	OUT_SetptQ					: REAL; 		(* (kVAr) Reactive power setpoint *)
	OUT_SetptQMax				: REAL;			(* (kVAr) Upper range of the Reactive Power setpoint*)
	OUT_SetptQMin				: REAL;			(* (kVAr) Lower range of the Reactive Power setpoint*)

	OUT_CmdReset				: BOOL ; 		(* (NA) Reset Command *) 
	
	MesHeartbeat				: BOOL ;		(*	NA) Heartbit of PCS*)
	MesCP_Read					: BOOL := TRUE;	(* (NA) CP to read values from PCS*)
	MesCP_Write					: BOOL := TRUE;	(* (NA) CP to write values from PCS*)
	
	
END_STRUCT
END_TYPE

// ---- 01_Equipement_Library/PCS/PCS_Sma.TcDUT
TYPE PCS_Sma :
STRUCT
		MesData					: PCS;		(* (NA) INV Struct*)
  	
	// System Parameter
		MesID_SystemState		:UINT; (* (-) Operating command for battery inverter, specified externally [AuxCtl.SCSOpCm d] *)
	
	// System Settings 
		MesID_CmdStopSystem		:UINT; (* (-) Disconnection of the inverter [FstStop] *)
		MesSetptQ_hldreg		:REAL; (* (%) Reactive power setpoint Q, in % of the maximum reactive power (with regard to VArRtg) of the inverter. [VArSpt] *)
		MesSetptP_hldreg		:REAL; (* (%) Active power setpoint P, in % of the maximum active power [WSpt] *)
	
	// inverter parameter
		MesID_CmdStop			:UINT; (* (-) Operating state of the inverter, setpoint [InvOpMod] *)
		MesErrClr				:UINT; (* (-) Acknowledgment of the present error [ErrClr] *)
		MesErrClrProErr			:UINT; (* (-) Acknowledging of safety-relevant errors [ErrClr.ProErr] *)
								
	// INV Measures 
		MesIdcStk1				:REAL; (* (A) DC current inverter bridge 1 [DcMs.Amp.Stk1] *)
		MesIdcStk2				:REAL; (* (A) DC current inverter bridge 2 [DcMs.Amp.Stk2] *)
		MesIdcStk3				:REAL; (* (A) DC current inverter bridge 3 [DcMs.Amp.Stk3] *)
		MesUdcStk1				:REAL; (* (V) DC voltage of the inverter bridge 1 [InvMs.DclVol.Stk1] *)
		MesUdcStk2				:REAL; (* (V) DC voltage of the inverter bridge 2 [InvMs.DclVol.Stk2] *)
		MesUdcStk3				:REAL; (* (V) DC voltage of the inverter bridge 3 [InvMs.DclVol.Stk3] *)
		MesIacL1				:REAL; (* (A) AC current L1, total [InvMs.TotA.PhsA] *)
		MesIacL2				:REAL; (* (A) AC current L2, total [InvMs.TotA.PhsB] *)
		MesIacL3				:REAL; (* (A) AC current L3, total [InvMs.TotA.PhsC] *)
		MesU12					:REAL; (* (V) Line-to-line voltage L1-L2, utility grid [GriMs.V.PhsAB] *)
		MesU23					:REAL; (* (V) Line-to-line voltage L2-L3, utility grid [GriMs.V.PhsBC] *)
		MesU31					:REAL; (* (V) Line-to-line voltage L3-L1, utility grid [GriMs.V.PhsCA] *)
		MesTmpAcCab				:REAL; (* (°C) Temperature in the AC range [TmpCab.Acc] *)
		MesTmpDcCab				:REAL; (* (°C) Temperature in the DC range [TmpCab.Dcc] *)
		MesTmpRioCab			:REAL; (* (°C) Temperature in the electronics area [TmpCab.Rio] *)
		MesTmpMax				:REAL; (* (°C) Temperature in interior, maximum value [TmpCab.Max] *)
		MesTmpIgbtMax			:REAL; (* (°C) Temperature of the inverter bridge (switch), maximum value [TmpStk.IgbtMax] *)
		MesTmpPcbMax			:REAL; (* (°C) Temperature of the inverter bridge (assembly), maximum value [TmpStk.PcbMax] *)
		MesTmpExt				:REAL; (* (°C) External temperature [TmpExl] *)
		MesTmpTransfo			:REAL; (* (°C) Temperature of the MV transformer [TmpTrf] *)
		MesID_SttDcSw1			:UINT; (* (-) Switching status of the DC load-break switch 1 [DcSw1Stt] *)
		MesID_SttDcSw2			:UINT; (* (-) Switching status of the DC load-break switch 2 [DcSw2Stt] *)
		MesID_SttDcSw3			:UINT; (* (-) Switching status of the DC load-break switch 3 [DcSw3Stt] *)
		MesID_SttAcSw			:UINT; (* (-) Switching status of the AC circuit breaker [AcSwStt] *)
		MesID_SttCapac			:UINT; (* (-) Switching state of the capacitor contactor [CapacSwStt] *)
		MesID_SttPrchrg			:UINT; (* (-) Switching status of the pre- charging contactor [PrchrgSwStt] *)
		MesEdcTot				:REAL; (* (MWh) DC energy drawn, total [Cnt.TotDcWhIn] *)
		MesEacTot				:REAL; (* (MWh) AC energy fed in, total [Cnt.TotAcWhOut] *)
		MesEdcDay				:REAL; (* (MWh) DC energy drawn that day [Cnt.DcWhIn] *)
		MesEacDay				:REAL; (* (MWh) AC energy fed in that day [Cnt.AcWhOut] *)
		MesID_ErrLcn			:UINT; (* (-) Error location of the present error [ErrLcn] *)
		MesID_ErrStt			:UINT; (* (-) Error status of the inverter [ErrStt] *)
		MesNum_Err				:UINT; (* (-) Error number of the present error [ErrNo] *)
		MesID_SttKey			:UINT; (* (-) Switch status of the start-stop key switch [Rio.KeySw] *) 
		MesTime_Feed			:UINT; (* (s) Feed-in time [Cnt.TotFeedTm] *)
		MesTime_Run				:UINT; (* (s) Operating time [Cnt.TotOpTm] *)
		MesTime_Fan1			:UINT; (* (s) Operating time of the interior fan 1 [Cnt.FanCab1Tm] *)
		MesTime_Fan2			:UINT; (* (s) Operating time of the interior fan 2 [Cnt.FanCab2Tm] *)
		MesTime_StkFan			:UINT; (* (s) Operating time of the inverter bridge fan [Cnt.FanStkTm] *)
		MesTime_Heater			:UINT; (* (s) Operating time of the interior heater [Cnt.HtCabTm] *)
		MesTime_Heater40C		:UINT; (* (s) Operating time of the -40°C interior heater [Cnt.HtLoExlTmpTm] *)
		MesTimeWait_Grid		:UINT; (* (s) Waiting time for grid connection [WaitGriTm] *)
		MesSerial				:UINT; (* (-) Inverter serial number [DevInf.SerNo] *)
		MesID_SttGfdi			:UINT; (* (-) Switching status of the GFDI [GfdiSwStt] *)
		MesSetptP				:REAL; (* (kW) Active power, setpoint [WSpt] *)
		MesSetptSmax			:REAL; (* (kVA) Maximum apparent power, setpoint [VAMaxSpt] *)
		MesSetptQ				:REAL; (* (kVAr) Reactive power, setpoint [VArSpt] *)
		MesCosPhisetpt			:REAL; (* (-) Power factor cos (phi), setpoint [PFSpt] *)
		MesID_SttPresTransfo	:UINT; (* (-) Fast stop hermetic protection, pressure [TrfPro.Pres] *)
		MesID_SttTempAlarmTransfo:UINT; (* (-) Fast stop hermetic protection, temperature [TrfPro.TmpTrp] *)
		MesID_SttOilAlarmTransfo:UINT; (* (-) Hermetic protection, gas fill level [TrfPro.GasOilLev] *)
		MesID_SttTempWarnTransfo:UINT; (* (-) Hermetic pressure, temperature warning [TrfPro.TmpWrn] *)
		MesTmpStk1				:REAL; (* (°C) Temperature of inverter bridge 1 (switch) [TmpStk1.lgbt] *)
		MesTmpStk2				:REAL; (* (°C) Temperature of inverter bridge 2 (switch) [TmpStk2.lgbt] *)
		MesTmpStk3				:REAL; (* (°C) Temperature of inverter bridge 3 (switch) [TmpStk3.lgbt] *)
		MesTmpStk1Max			:REAL; (* (°C) Maximum temperature of inverter bridge 1 (assembly) [TmpStk1.Pcb] *)
		MesTmpStk2Max			:REAL; (* (°C) Maximum temperature of inverter bridge 2 (assembly) [TmpStk2.Pcb] *)
		MesTmpStk3Max			:REAL; (* (°C) Maximum temperature of inverter bridge 3 (assembly) [TmpStk3.Pcb] *)
		MesEacPrevDay			:REAL; (* (MWh) AC energy fed in the previous day [Cnt.YstdWhOut] *)
		MesTime_CPU				:REAL; (* (s) CPU running time since system start [Cpu1UpTime] *)
		MesRiso					:REAL; (* (kOhm) Insulation resistance [PvGnd.RisIso] *)
		MesPressureTransfo		:REAL; (* (-) MV transformer pressure [PresTrf] *)
		MesID_SttPressureSensor	:UINT; (* (-) Error status of MV transformer pressure monitoring [PresTrf.ErrStt] *)
		MesSetptPmax			:REAL; (* (pu) Available Active Power [WAval] *)
		MesSetptQmax			:REAL; (* (pu) Available reactive power [VArAval] *)
		MesID_SttDrt			:UINT; (* (-) Current derating status [DrtStt] *)
		MesID_PwrOffReas		:UINT; (* (-) Current cause of inverter disconnection [PwrOffReas] *)
		MesPnom_stpt			:REAL; (* (kW) Nominal value of active power [WRtg] *)
		MesActErrNo1			:UINT; (* (-) Error number of the current error [ActErrNo1] *)
		MesActErrLcn1			:UINT; (* (-) Location where the current error was detected [ActErrLcn1] *)
		MesActErrNo2			:UINT; (* (-) Error number of the current error [ActErrNo2] *)
		MesActErrLcn2			:UINT; (* (-) Location where the current error was detected [ActErrLcn2] *)
		MesActErrNo3			:UINT; (* (-) Error number of the current error [ActErrNo3] *)
		MesActErrLcn3			:UINT; (* (-) Location where the current error was detected [ActErrLcn3] *)
		MesActErrNo4			:UINT; (* (-) Error number of the current error [ActErrNo4] *)
		MesActErrLcn4			:UINT; (* (-) Location where the current error was detected [ActErrLcn4] *)
		MesActErrNo5			:UINT; (* (-) Error number of the current error [ActErrNo5] *)
		MesActErrLcn5			:UINT; (* (-) Location where the current error was detected [ActErrLcn5] *)
		MesActErrNo6			:UINT; (* (-) Error number of the current error [ActErrNo6] *)
		MesActErrLcn6			:UINT; (* (-) Location where the current error was detected [ActErrLcn6] *)
		MesActErrNo7			:UINT; (* (-) Error number of the current error [ActErrNo7] *)
		MesActErrLcn7			:UINT; (* (-) Location where the current error was detected [ActErrLcn7] *)
		MesActErrNo8			:UINT; (* (-) Error number of the current error [ActErrNo8] *)
		MesActErrLcn8			:UINT; (* (-) Location where the current error was detected [ActErrLcn8] *)
		MesActErrNo9			:UINT; (* (-) Error number of the current error [ActErrNo9] *)
		MesActErrLcn9			:UINT; (* (-) Location where the current error was detected [ActErrLcn9] *)
		MesActErrNo10			:UINT; (* (-) Error number of the current error [ActErrNo10] *)
		MesActErrLcn10			:UINT; (* (-) Location where the current error was detected [ActErrLcn10] *)
		MesQref_stptExt			:REAL; (* (kVAr) Reference value for the external reactive power setpoint [VArExlSpt.RefVal] *)
		MesPref_stptExt			:REAL; (* (kW) Reference value for the external active power setpoint [WExlSpt.RefVal] *)
		ModbusValue 			:WORD;
		MesQref_stpt			:REAL; (* (kvar) Nominal value of reactive power [VArRtg] *)
		MesUdc_plusGnd			:REAL; (* (V) DC voltage of DC+ to ground [DcMs.VolPosGnd] *)
		MesUdc_minusGnd			:REAL; (* (V) DC voltage of DC- to ground [DcMs.VolNegGnd] *)
		MesID_State_Imax		:UINT; (* (-) Overload capability: Overcurrent status [GriForm.OvAmpStt] *)
		MesTimeWait_Error		:REAL; (* (s) Remaining error waiting period [ErrRmgTm] *)
		
	// State ID 
		MesID_OpeMode			: WORD ; (* SMA Operating Mode  ENUM *)
		MesID_OpStt				: WORD ; (* SMA Operation State ENUM *)
		MesID_OpeProErr			: WORD ; (* SMA Saftey Error  ENUM *)
		MesID_ErrClr			: WORD ; (* SMA Error ENUM *)

	// Output 
		OUT_CmdReset_Safety		: BOOL ;(* Safety reset ordered *) 
		OUT_CmdOpenAC			: BOOL ; (* Open AC Command*)
END_STRUCT
END_TYPE

// ---- 01_Equipement_Library/PCS/PCS_Jema_IBX3.TcDUT
///////////
// Structure for CtrlPcs Jema .  
//////////
TYPE PCS_Jema_IBX3 :
STRUCT
// PCS Controller  Measures
	AX_PowerCol					: ARRAY[1..3] OF PowerCol_Jema;

	MesData						: PCS ; 
	
	
	MesNbPowerCol_FreqReg			: UINT  ; (*(NA) Number of Power Column doing frequency regulation *)
	MesState_SoCLimitReached		: BOOL ; (*(NA) PCS SoC Limits has been reached *)
	MesHumidity						: REAL ; (*(%) Humidity*)
	
	MesReadCompleted				: BOOL ; 
	
	OUT_CmdBlackStart			: BOOL ; (* (NA) Blackstart Command *) 
	OUT_CmdGridMode				: BOOL ; (* (NA) Grid Mode Command *) 
	OUT_CmdP					: BOOL ; (* (NA) P setpoint regulation Mode Command *) 
	
	OUT_CmdQ				: BOOL ; (* (NA) Q setpoint regulation Mode Command *) 
	OUT_SetptV				: REAL ; (* (V) Voltage Reference for offgrid Mode *) 
	OUT_SetptCosPhi			: REAL ; (* (p.u) Cosphi Reference for Cosphi reg Mode *) 
	
	OUT_SetptF				: REAL ; 	(* (Hz) Frequency Reference for offgrid Mode *) 
	OUT_CmdCosPhi			: BOOL ; (* (NA) Cosphi regulation Mode Command *) 
	OUT_CmdUregMode			: BOOL ; (* (NA) Voltage Regulation Mode Command *) 
	OUT_CmdFreqregMode	: BOOL ; (* (NA) Frequency Regulation Mode Command *) 
END_STRUCT
END_TYPE

// ---- 01_Equipement_Library/PCS/PCS_PE.TcDUT
{attribute 'pack_mode' := '1'}
TYPE PCS_PE :
STRUCT
// PCS Controller  Measures
	AX_PowerCol					: ARRAY[1..6] OF PowerCol_PE;		(* PE Module*)
	
	MesData						: PCS ; (* MesData*)
	
	MesP_ChargeMax				: REAL ;		(* (%)	Max active power setpoint. SV4.2.1a	*)
	MesP_DischargeMax			: REAL ;		(* (%)	Max active power setpoint. SV4.2.1b	*)
	MesP_ChargeMax1				: REAL ;		(* (%)	Max active power setpoint1. SV4.2.1a	*)
	MesP_DischargeMax1			: REAL ;		(* (%)	Max active power setpoint1. SV4.2.1b	*)
	MesP_ChargeMax2				: REAL ;		(* (%)	Max active power setpoint2. SV4.2.1a	*)
	MesP_DischargeMax2			: REAL ;		(* (%)	Max active power setpoint2. SV4.2.1b	*)
	
	//Electrical Measurements	
	MesI1						: REAL; (* (A) Current phase 1 (R). INV: SV1.4 Grid current I1 (HEMK)															*)
	MesI2						: REAL; (* (A) Current phase 2 (S). INV: SV1.5 Grid current I2 (HEMK)															*)
	MesI3						: REAL; (* (A) Current phase 3 (T). INV: SV1.6 Grid current I3  (HEMK)															*)
	MesU12						: REAL; (* (V) Phase AB RMS voltage (line to line)at grid side of AC circuit breaker CB501. INV: SV1.1 Grid voltage RS (HEMK)	*)
	MesU23						: REAL; (* (V) Phase BC RMS voltage (line to line)at grid side of AC circuit breaker CB501. INV: SV1.2 Grid voltage ST(HEMK)	*)
	MesU31						: REAL; (* (V) Phase CA RMS voltage (line to line)at grid side of AC circuit breaker CB501. INV: SV1.3 Grid voltage TR (HEMK)	*)

	MesHumidity					: REAL;			(* (%) Humidity sensor	*)
	MesPconnected				: REAL; (* (%) Current available active power. INV: SV4.1.2 P limit inst 														*)  
	MesQconnected				: REAL; (* (%) Current available reactive power. INV: SV4.2.2 Q limit inst 														*)                                                      									

	MesIDState_InsuResistor_DC	: WORD ; (* (NA) Status of insulation protection. 0 = Idle, 1= Inter measurement quard, 2=measurement in progress, 3=self-test in progress, 4=risk addressed state SV3.1.1 *)
	MesInsuResistor_AC			: REAL;	(* (Ohms) AC Insulation Resistance. INV: SV3.1.2  Resistor 																*)
	MesIDState_InsuResistor_AC	: WORD ; (* (NA) Status of insulation protection. 0 = Idle, 1= Inter measurement quard, 2=measurement in progress, 3=self-test in progress, 4=risk addressed state SV3.1.1 *)
	MesInsuResistor_DC			: REAL;	(* (Ohms) DC Insulation Resistance. INV: SV3.2.2  Resistor 		*)
	MesInsuResistor_DC2			: REAL; (* (Ohms) DC Insulation Resistance. INV: SV3.3.2  Resistor 		*)

	MesUdc_Input1		 		: REAL ; (* (V) DC Voltage Bus 1 . INV : SV2.1.1 *)
	MesUdc_Input2		 		: REAL ; (* (V) DC Voltage Bus 2 . INV : SV2.1.2*)
	MesUdc_Input3		 		: REAL ; (* (V) DC Voltage Bus 3 . INV : SV2.1.3*)
	MesUdc_Bat1		 			: REAL ; 	(* (V) DC Voltage BESS 1 . INV : SV2.4.1*)
	MesUdc_Bat2		 			: REAL ; 	(* (V) DC Voltage BESS 2 . INV : SV2.4.2*)
	MesUdc_Bat3		 			: REAL ; 	(* (V) DC Voltage BESS 3 . INV : SV2.4.3*)
	MesPdc_Input1		 		: REAL ; (* (V) DC Power Bus 1 . INV : SV2.5a*)
	MesPdc_Input2		 		: REAL ; (* (V) DC Power Bus 2 . INV : SV2.5b*)
	MesPdc_Input3		 		: REAL ; (* (V) DC Power Bus 3 . INV : SV2.5c*)
	MesIdc_RFI_Input1    		: REAL ; (* (V) RFI Current  Bus 1 . INV : SV2.11a*)
	MesIdc_RFI_Input2    		: REAL ; (* (V) RFI Current  Bus 2 . INV : SV2.11b*)
	MesIdc_RFI_Input3	 		: REAL ; (* (V) RFI Current  Bus 3 . INV : SV2.11c*)
	MesIdc_Input1				: REAL; (*(A) SV2.6a DC input current*)
	MesIdc_Input2				: REAL; (*(A) SV2.6b DC input current*)
	MesIdc_Input3				: REAL; (*(A) SV2.6c DC input current*)

	//Status Summary
	MesIDState					: UINT; (* (NA) Current inverter status . INV : SV4.1.3                                                    *)                 	
	MesAlarmID					: WORD;	(* (NA) Alarm ID of the currently active event.  INV : SV4.1.1    *)
	MesWarningID				: WORD;	(* (NA) Warning ID of the currently active event.  INV : SV4.1.2    *)
	MesEventID					: WORD;	(* (NA) Event ID of the currently active event.  INV : SV9.1.1 :Last Event    *)
                    	
	// Inverter's Control Cabinet  Status                                                                       											
	MesTemp_IGBTmax				: REAL; 		 (* (C) Maximum IGBT temperature. INV: SV4.1.5 Max IGBTs temperature											*)
	MesTemp_PowerColmax			: REAL; 		 (* (C) Maximum power column temperature. INV: SV4.1.6 Max modules temperature									*)
 
	MesReadModule				: UINT;		(* (NA) module read *)
	MesIDState_PowerCol			: WORD ; 	(* (NA) Running modules (0 = stopped, 1 =running). Module 1 is the first from the right. SV9.1.1															*)
               	                                                   	                                						
	// Reset command        	                                                                     	                                						
	OUT_CmdReset 				: BOOL; 		 (* (NA) OUT reset command. INV: Reset command 43012															*)
	MesCalibrationState		 	: WORD;			(*(NA) it's a state to know if the calibration is ongoing or not, (0=running, 1=Discharging the batteries started, 2=20min hold finished, starting to send setpt of 0 for 20min, 3=Charging started*)
	MesBMSSelected				: WORD;
	OUT_SetptPMax_IMDicharge1	: REAL;
	OUT_SetptPMax_IMDicharge2	: REAL;
	OUT_SetptPMax_IMCharge1		: REAL;
	OUT_SetptPMax_IMCharge2		: REAL;
	MesSelector 				: BOOL;
	
	
END_STRUCT
END_TYPE

// ---- 01_Equipement_Library/PCS/PowerCol_JemaAlarms.TcDUT
TYPE PowerCol_JemaAlarms :
STRUCT

// ALARM0 bAlarm1
		MesI1_Alm			: BOOL; 	//RegAlarms0: I1_Alm
		MesI2_Alm			: BOOL; 	//RegAlarms0: I2_Alm
		MesI3_Alm			: BOOL; 	//RegAlarms0: I3_Alm
		MesVdc_High_Alm		: BOOL; 	//RegAlarms0: Vdc_High_Alm
		MesVdc_Low_Alm		: BOOL; 	//RegAlarms0: Vdc_Low_Alm
		                            	// 
		MesU12_High_Alm		: BOOL; 	//RegAlarms0: U12_High_Alm
		MesU12_Low_Alm		: BOOL; 	//RegAlarms0: U12_Low_Alm
		MesU23_High_Alm		: BOOL; 	//RegAlarms0: U23_High_Alm
		MesU23_Low_Alm		: BOOL; 	//RegAlarms0: U23_Low_Alm
		MesU31_High_Alm		: BOOL; 	//RegAlarms0: U31_High_Alm
		MesU31_Low_Alm		: BOOL; 	//RegAlarms0: U31_Low_Alm
		MesVd_High_Alm		: BOOL; 	//RegAlarms0: Vd_High_Alm
		MesVd_Low_Alm		: BOOL; 	//RegAlarms0: Vd_Low_Alm
		MesVdc_Neg			: BOOL; 	//RegAlarms0: Vdc_Neg
		                            	//   :blabla
										//wAlarmCode
		
// ALARM1 bAlarm1
		MesU1223_Unbalance	: BOOL;		//RegAlarms1: U1223_Unbalance
		MesU2331_Unbalance	: BOOL;		//RegAlarms1: U2331_Unbalance
		MesU3112_Unbalance	: BOOL;		//RegAlarms1: U3112_Unbalance
		MesInvertedPhase	: BOOL;		//RegAlarms1: InvertedPhase
		MesI12_Unbalance	: BOOL;		//RegAlarms1: I12_Unbalance
		MesI23_Unbalance	: BOOL;		//RegAlarms1: I23_Unbalance
		MesI31_Unbalance	: BOOL;		//RegAlarms1: I31_Unbalance
		MesCouplingTimeout	: BOOL;		//RegAlarms1: CouplingTimeout
		MesF_High			: BOOL;		//RegAlarms1: F_High
		MesF_Low			: BOOL;		//RegAlarms1: F_Low
		MesGrndFault		: BOOL;		//RegAlarms1: GrndFault
		MesVaristor			: BOOL;		//RegAlarms1: Varistor
		MesPcbOverTemp		: BOOL;		//RegAlarms1: PcbOverTemp
		MesHeatsinkOverTemp	: BOOL;		//RegAlarms1: HeatsinkOverTemp
		                           		// 
		MesOvertempHyst		: BOOL;		//RegAlarms1: OvertempHyst
		//wAlarmCode
// ALARM2 bAlarm1
										// 
                                    	// 
                                    	// 
                                    	// 
		MesGridCbOpened		: BOOL;		//RegAlarms2: GridCbOpened
		MesGridCbTrip		: BOOL;		//RegAlarms2: GridCbTrip
										//
		                           		// 
		MesGridContactFail	: BOOL;		//RegAlarms2: GridContactFail 
		MesDoorOpened		: BOOL;		//RegAlarms2: DoorOpened 
		                           		// 
		                           		// 
		MesVdcPrechargewrong: BOOL;		//RegAlarms2: VdcPrechargewrong 
		                           		// 
		MesOverVoltHyst		: BOOL;		//RegAlarms2: OverVoltHyst 
		MesIdcMax			: BOOL;		//RegAlarms2: IdcMax 
		//wAlarmCode
		
//ALARM3   bAlarm1                         
		MesSKIIP1			: BOOL; 	//RegAlarms3: SKIIP1
		MesSKIIP2			: BOOL; 	//RegAlarms3: SKIIP2
		MesSKIIP3			: BOOL; 	//RegAlarms3: SKIIP3
		MesSKIIP_OT			: BOOL; 	//RegAlarms3: SIIP_OT
		MesFPGA_WdogTrip	: BOOL; 	//RegAlarms3: FPGA_WdogTrip
		MesStopEverything	: BOOL; 	//RegAlarms3: StopEverything
		MesIMax				: BOOL; 	//RegAlarms3: IMax
		MesEmergencyStop	: BOOL; 	//RegAlarms3: EmergencyStop
		MesImdWarning		: BOOL; 	//RegAlarms3: ImdWarning
		MesImdFault			: BOOL; 	//RegAlarms3: ImdFault
		                            	//RegAlarms3:  
		MesCoilOverTemp		: BOOL; 	//RegAlarms3: CoilOverTemp
		                            	//RegAlarms3:  
		MesAlrmGrp1_Curr	: BOOL; 	//RegAlarms3: AlrmGrp1_Curr
		MesAlrmGrp2_Curr	: BOOL; 	//RegAlarms3: AlrmGrp2_Curr
		MesShortCircuit_DC	: BOOL; 	//RegAlarms3: ShortCircuit_DC
		//wAlarmCode
// ALARM4 bAlarm1
		MesBatError			: BOOL;		//RegAlarms4: BatError
		MesBatCtlStop		: BOOL;		//RegAlarms4: BatCtlStop
		MesBatComErrors		: BOOL;		//RegAlarms4: BatComErrors
		MesPowerUnbalance	: BOOL;		//RegAlarms4: PowerUnbalance
		MesOverpower		: BOOL;		//RegAlarms4: Overpower
		//wAlarmCode
		
END_STRUCT
END_TYPE

// ---- 01_Equipement_Library/PCS/PowerCol_Jema.TcDUT
///////////
// Structure For Jema Module 
//////////
TYPE PowerCol_Jema :
STRUCT
	
		MesData					: PowerCol ; (* MesData *) 

		MesTempControl      		: REAL ; 		// {0}(°C) Temperature of control card
		MesTempPowerUnit    		: REAL ;		// {0}(°C) Temperature of Power Unit
		MesTempCabinet      		: REAL ; 		// {0}(°C) Cabinet temperature
		MesTempCoil1        		: REAL ; 		// {0}(°C) Coil temperature
		MesRegAlarm0        		: WORD ; 		// {0}Alarm Word of PCS
		MesRegAlarm1        		: WORD ; 		// {0}Alarm Word of PCS 
		MesRegAlarm2        		: WORD ; 		// {0}Alarm Word of PCS 
		MesRegAlarm3        		: WORD ;  		// {0}Alarm Word of PCS
		MesRegAlarm4        		: WORD ;  		// {0}Alarm Word of PCS
		MesDeratingWord				: WORD ;		// {0}Derating word of PCS
		MesHeartbit					: REAL ;		// {0}Heartbit
		MesDoorOpened				: BOOL ;		// {1}Door of the Power module is opened	
		
		MesJemaAlarms				: PowerCol_JemaAlarms;

			

END_STRUCT
END_TYPE

// ---- 01_Equipement_Library/PCS/PowerCol.TcDUT
///////////
// Structure For Jema Module 
//////////
TYPE PowerCol :
STRUCT
		MesP 						: REAL; 		// {1}(kW) Active Power output (AC) of PCS
		MesQ 						: REAL; 		// {1}(kVAr) Reactive AC Power Produced by PCS 
		MesPdc						: REAL ; 		// {1}(kW) DC Power . 
		MesCosPhi 					: REAL;  		// {0}(p.u) Power factor
		MesFreq						: REAL ; 		// {0}(Hz) Frequency
		MesTemp						: REAL ; 		// {0}(°C) PCS Internal Temperature
		MesU 						: REAL;  		// {0}(V) AC Voltage measure
		MesUdc 						: REAL;  		// {0}(V) DC Voltage measure
		MesI 						: REAL; 		// {0}(A) Total AC current 
		MesI1						: REAL ; 		// {0}(A) Phase 1 AC Current
		MesI2						: REAL ;        // {0}(A) Phase 2 AC Current
		MesI3						: REAL ;        // {0}(A) Phase 3 AC Current
		MesIdc 						: REAL; 		// {0}(A) Total DC current from batteries (+ = discharge)
		MesPavailable 				: REAL;  		// {1}(kW) Available PCS Power 
		MesPconnected				: REAL ; 		// {0}(kW) Connected PCS Power 
		MesDcSwitchClosed			: BOOL ; 		// {0}(NA) Position of the DC Switch : True = Switch closed
		MesAcSwitchClosed			: BOOL ; 		// {0}(NA) Position of the AC Switch : True = Switch closed
	

			

END_STRUCT
END_TYPE

// ---- 01_Equipement_Library/PCS/PowerCol_PE.TcDUT
///////////
// Structure For Jema Module 
//////////
TYPE PowerCol_PE :
STRUCT
		
		MesData					: PowerCol ; (* MesData *) 

		AX_DCInputs			: ARRAY[1..10] OF  DCInputs_PE ;(* Object *) 
		
		MesIDState			: DWORD ;		(* (NA) 	Module status (SV9.3 PE documentation p.97)																*)
		MesTempmax			: REAL ;		(* (C) 		Maximum IGBT temperature of the selected module															*)
		MesStateIO			: WORD ;		(* (NA) 	0: Open, 1: Closed. Bit 1 =  fan contactor, Bit 2 = main AC contactor, Bit 3 = AC soft charge contactor, Bit 4 = LCL filter contactor, Bit 5 = DC contactor , Bit 6 = reserved, Bit 7 = if open : overheating in the coil, Bit 8 = fan contactor feedback, Bit 9 = AC main contactor feedback, Bit 10 = AC soft charge contactor feedback, Bit 11 = LCL filter contactor feedback , Bit 12 = DC contactor feedback *) 		
		MesHygro			: REAL ; 		(* (%) 		Percentage of humidity																					*)
		MesAlarmID			: BYTE ; 		(* (NA)  PowerColumn Alarm ID  . W65 to W116  *)
			

END_STRUCT
END_TYPE

// ---- 01_Equipement_Library/PPC/PPC.TcDUT
///////////
// Structure For Inverter. Main Operating Data to be saved ( ex: OPC ) .  
//////////
TYPE PPC :
STRUCT
	
		// INV Measures
		
		MesAlarmCom					: BOOL; 		(* (NA) PPC  Communication fault*)
		

		
		MesSetptP			: REAL;
		MesSetptQ			: REAL;		
		MesP				: REAL;
		MesQ				: REAL;

		MesNbInvAvail		: REAL;


		
		MesWatchdog			: REAl;
		CalState			: BYTE;
		
		MesCP_Read			: BOOL := TRUE;	(* (NA) Cal : Permanent Condition for Read			  *)
		MesCP_Write			: BOOL := FALSE;(* (NA) Cal : Permanenent Condition for Write	  	  *)
		   
		MesAlarmCode		: WORD ;    (* (NA) Internal Akuo AlarmCode*)
		MesWarningCode		: WORD ;    (* (NA) Internal Akuo WarningCode*)
		MesEventCode		: WORD ;    (* (NA) Internal Akuo EventCode*)
		
END_STRUCT
END_TYPE

// ---- 01_Equipement_Library/PPC/PPC_Sma.TcDUT
///////////
// Structure For Inverter. Main Operating Data to be saved ( ex: OPC ) .  
//////////
TYPE PPC_Sma :
STRUCT
	
		// INV Measures
		MesData		: PPC ; 
		
		
		MesPState			: REAL;
		MesQState			: REAL;
		MesGeneState		: REAL;

		MesPNomControlled	: REAL;
		MesPControlled		: REAL;
		MesQnomControlled	: REAL;
		MesQControlled		: REAL;
		
		
END_STRUCT
END_TYPE

// ---- 01_Equipement_Library/PPC/PPC_PE.TcDUT
TYPE PPC_PE :
STRUCT
		MesData 								: PPC;   			    (* (NA) MesData				 *)
		                                                                
		PM										: PM_PM5XXX;	    (* (NA) PM13EH PLUS			 *)
		EL3453									: PM_Standard;		    (* (NA) Beckhoff card EL3453 *)
		MesState								: UINT;				    (* (NA) PPC status. 0: PPC off and not sending commands to inverters, 1: PPC on and sending commands to inverters, 2: PPC on frequency event. 3: PPC in LVRT event. 4: PPC in HVRT event. 5, 6: Reserved *)
                                                                        	                                                            
		// Q Regulation                                                                                                                                            		    		
		ParamQfUQmin							: REAL := -5000;	    (* (kVAr) Voltage Regulation Minimal Reactive Power @ maximal voltage*) 		
		ParamQfUQmax							: REAL := 5000;  	    (* (kVAr) Voltage Regulation Maximal Reactive Power @ minimal voltage*)    		
		ParamQfUUHigh							: REAL := 25000; 	    (* (V)    Voltage Regulation Maximal voltage*)    		
		ParamQfUDdBandHigh						: REAL := 22000; 	    (* (V)    Voltage Regulation Deadband High voltage*)     		
		ParamQfUDdBandLow						: REAL := 18000; 	    (* (V)    Voltage Regulation Deadband Low voltage*)      	
		ParamQfUULow							: REAL := 15000; 	    (* (V)    Voltage Regulation Minimal Voltage*)
		MesAlarmPower							: BOOL; 				(* (NA)   Power alarm due to circuit breaker open										 						*)			
                                                                                                                                                			 							
	// PI active power                                                                                                                          			 							
		//IN_CmdPIDP_LocalMode 					: BOOL;                                                                                         			 							
		IN_SetptP_PR_Cent						: REAL;					(* (%)  Active power reference  														 						*)
		IN_SetptP_PR_MW							: REAL;					(* (MW) Active power reference 														 							*)	
		IN_Feedback_PR_Cent						: REAL;					(* (%)	Active power PI feedback 													 							*)
		IN_Feedback_PR_MW						: REAL;					(* (MW)	Active power PI feedback 													 							*)
		MesStateOL_PR							: BOOL;					(* (NA) Open loop activation of P control. 1= Open loop activated					 							*)
		IN_PIDP_SetptPOpenloop					: REAL;		            (* *)                            	                                    			 							                                                              			 
		ParamKp_PR								: REAL;					(* (NA) Kp for P regulation 														 							*)
		ParamKi_PR								: REAL;					(* (NA) Ki for P regulation 	 													 							*)
	   	ParamPIDP_Inversion						: BOOL;					(* (NA) PI inversion of active power control 										 							*)    
		ParamPID_PR_Min							: REAL; 				(* (kW) Low limit for PI for active power regulation	   							 							*)     		
		ParamPID_PR_Max							: REAL;  				(* (kW) High limit for PI for active power regulation 								 							*)          		
	    OUT_SetpointP_PR						: REAL;					(* (p.u) Active Power PI output per unit 											 							*)                                                                                                                                       			 
	
// PI frequency control                                                                                                                     			 							
		IN_SetptFreq_FR_Unit					: REAL;					(* (p.u) Frequency regulation (FR) reference  										 							*)
		IN_SetptFreq_FR_MW						: REAL;					(* (MW) Frequency regulation (FR) reference 										 							*) 
		IN_Feedback_FR_Unit						: REAL;					(* (p.u) Frequency regulation (FR) PI feedback 										 							*)
		IN_Feedback_FR_MW						: REAL;					(* (MW)	Frequency regulation (FR) PI feedback 										 							*)	
        ParamKp_FR								: REAL;					(* (NA) Kp for frequency regulation													 							*)
		ParamKi_FR								: REAL;					(* (NA) Ki for frequency regulation 		 										 							*)
	    ParamFreqnom							: REAL;					(* (NA) Nominal frequency for frequency response									 							*) 
		ParamStatism_OverFreq_Primary			: REAL; 				(* (NA) Slope for the Primary point Over Frequency in Frequency Response			 							*) 
		ParamStatism_OverFreq_Secundary			: REAL;					(* (NA) Slope for the Secundary point Over Frequency in Frequency Response 			 							*)
        ParamStatism_UnderFreq_Primary			: REAL; 				(* (NA) Slope for the Primary point under Frequency in Frequency Response			 							*) 
		ParamStatism_UnderFreq_Secundary		: REAL;					(* (NA) Slope for the Secundary point under Frequency in Frequency Response 		 							*)
		ParamDeltaPmax_OverFR					: REAL; 				(* (kW) Maximum power to be injected during under frequency regulation 		 		 							*)
        ParamDeltaPmax_UnderFR					: REAL; 				(* (kW) Maximum power to be reduced during over frequency regulation 		 		 							*)
		ParamDeadBand_FR						: REAL;					(* (mHz) Frequency regulation dead band axis Y										 							*) 
		MesEventID_FR							: UINT;					(* (NA) Frequency Response Event State. 0: No Event, 1: Over Frequency Primary Band, 2: Over Frequency Secondary Band, 3: Over Frequency Terciary Band, 4: Under Frequency Primary Band, 5: Under Frequency Secondary Band, 6: Under Frequency Terciary Band *)
 		MesStateID_FR							: BOOL;					(* (NA) Frequency Mode Selector. Calculation basis: 0: unitary base, 1: Power freeze 							*)		
		MesState_FR								: BOOL;					(* (NA) Activation/deactivation of frequency regulation. 1= activated				 							*)
		                               
	// PID Q direct                               	
		IN_SetptQ_QR_Cent					    : REAL;					(* (%) Reactive power reference  													 							*)
		IN_SetptQ_QR_MW							: REAL;					(* (MVAr) Reactive power reference 													 							*)	
		IN_Feedback_QR_Cent						: REAL;					(* (%) Reactive power PI feedback 													 							*)
		IN_Feedback_QR_MW						: REAL;					(* (MVAr) Reactive power PI feedback 												 							*)
		MesStateOL_QR							: BOOL;					(* (NA) Open loop activation of Q control. 1= Open loop activated					 							*)
		ParamKp_QR								: REAL;					(* (NA) Kp pour régulation Q 										 				 							*)
		ParamKi_QR								: REAL; 				(* (NA) Ki pour régulation Q 														 							*)
 		ParamPID_QR_Min							: REAL; 				(* (kVAr) Low limit for PID of reactive Power  										 							*)     		
		ParamPID_QR_Max							: REAL;  				(* (kVAr) High limit for PID of active Power										 							*)
		ParamPIDQ_Inversion						: BOOL;					(* (NA) PI inversion of RPCF control												 							*)  
		OUT_SetpointQ_QR						: REAL;					(* (p.u) Reactive Power PI output per unit 											 							*)
		
	// Cos(phi)
		ParamCosPhiMax							: REAL;				    (* (p.u)TanPhi Max limit for Q regulation																		*)
		ParamCosPhiMin							: REAL;				    (* (p.u)TanPhiMin limit for Q regulation 																		*)
		ParamCosPhiLagging						: BOOL;				    (* (NA) Lagging/inductive [soutirer]= 1: Q absorption Q-.  Leading/Capacitive = 0: Q injection Q+ 				*)
		ParamCosPhi								: REAL; 				(* (p.u) Desired cosPhi setpoint 																				*)                                                                
		MesState_PFR							: BOOL;				    (* (NA) CosPhi Regulation is activated	     																	*)
		MesSetptCosPhi							: REAL;				    (* (p.u) Measured setpoint Cos Phi				 																*)
		ParamKp_PFR								: REAL;					(* (NA) Kp for cos(phi) regulation													 							*)
		ParamKi_PFR								: REAL; 				(* (NA) Ki for cos(phi) regulation										 			 							*)
 		ParamPID_PFR_Min						: REAL; 				(* (kVAr) Low limit for PID of cos(phi) regulation  								 							*)     		
		ParamPID_PFR_Max						: REAL;  				(* (kVAr) High limit for PID of cos(phi) regulation									 							*)
		ParamPID_PFR_Inversion					: BOOL;					(* (NA) PI inversion of cos(phi) regulation											 							*)  
		OUT_Setpoint_PFR						: REAL;					(* (p.u) cos(phi) regulation PI output per unit 											 					*)
		
	// V regulation
		IN_SetpointV_VR_kV						: REAL;					(* (kV) Voltage reference																						*)
		IN_SetpointV_VR_Cent					: REAL; 				(* (%) Voltage reference																						*)                                                                
		IN_Feedback_VR_Cent						: REAL;					(* (%) Voltage PI feedback 													 									*)
		IN_Feedback_VR_kV						: REAL;					(* (kV) Voltage PI feedback 												 									*)
		
		ParamKp_VR								: REAL;					(* (NA) Kp for voltage regulation													 							*)
		ParamKi_VR								: REAL; 				(* (NA) Ki for voltage regulation										 			 							*)
 		ParamPID_VR_Min							: REAL; 				(* (kV) Low limit for PID of voltage regulation  								 								*)     		
		ParamPID_VR_Max							: REAL;  				(* (kV) High limit for PID of voltage regulation									 							*)
    	ParamPID_VR_Inversion					: BOOL;					(* (NA) PI inversion of voltage regulation											 							*)  
		OUT_Setpoint_VR							: REAL;					(* (p.u) Voltage regulation PI output per unit 											 						*)
		ParamStatism_V_VR						: REAL; 				(* (NA) Droop V for voltage regulation 			 																*) 
		ParamStatism_Q_VR						: REAL; 				(* (NA) Droop Q for voltage regulation 			 																*)
	
	// Q(V)
		IN_SetpointQ_QRV_Cent					: REAL; 				(* (%) Q(V) reference																							*)                                                                
		IN_Feedback_QRV_Cent					: REAL;					(* (%) Q(V) PI feedback 													 									*)
		MesSetptQ_QRV							: REAL;				    (* (p.u) Measured Q setpoint for Q(V)			 																*)
		ParamKp_QRV								: REAL;					(* (NA) Kp for Q(V)																	 							*)
		ParamKi_QRV								: REAL; 				(* (NA) Ki for Q(V)														 			 							*)
 		ParamPID_QRV_Min						: REAL; 				(* (kV) Low limit for PID of Q(V)				  								 								*)     		
		ParamPID_QRV_Max						: REAL;  				(* (kV) High limit for PID of Q(V)													 							*)
    	ParamPID_QRV_Inversion					: BOOL;					(* (NA) PI inversion of Q(V)														 							*)  
		OUT_Setpoint_QRV						: REAL;					(* (p.u) Reactive power depending of Voltage output per cent							 						*)

// Regulation status and modes
		MesLocalMode							: BOOL; 			    (* (NA) In Local mode, the DEIE is inhibated  																	*)
		
		MesIDState_QReg							: UINT;				    (* (NA) Q control selection. 0: no Q control. 1: Q_ref / RPCF. 2: Reserved. 3: cos(phi) control. 4: VRS control. 5: PF - VRS. 6: cos-phi(P). 7: Q(V). 8: dQ(V). 9: dQ(eV). 10: Reserved *)                                                   
		MesState_PR								: BOOL;					(* (NA) Enabling of P_REF control		  *)
		MesState_PRDelta						: BOOL;					(* (NA) Enabling of P_delta control		  *)
		CmdState_FR								: BOOL;					(* (NA) Enabling of freq response control *)
		CmdState_PR								: BOOL;					(* (NA) Enabling of P_REF control		  *)
		MesState_QR 							: BOOL;					(* (NA) Q_reference control selection. WS only *)
		CmdState_PFR							: BOOL;					(* (NA)  COS(phi) control selection. WS only *)
		MesState_VRS							: BOOL;					(* (NA) VRS control selection. WS only *)
		MesState_PFRP							: BOOL;					(* (NA) cosphi(P) control selection. WS only *)
		MesState_QRV							: BOOL;					(* (NA) Q(V) control selection. WS only *)
		MesState_QRamp							: BOOL;					(* (NA) Q ramps. 1 enable, 0 disable *)
		MesState_PRamp							: BOOL;					(* (NA) P ramps. 1 enable, 0 disable *)
	    MesState_PQPriority						: BOOL;					(* (NA) Status. 0: No priority acting, 1: P priority acting, 2: Q priority acting *)
		MesPlimit_PQPriority					: BOOL;					(* (NA) P REFERENCE LIMIT due TO PQ priority in p.u. *)
		MesQlimit_PQPriority					: BOOL;					(* (NA) Q reference limit due to PQ priority in p.u. *)
		
		MesPnom									: REAL;					(* (kW) Defined nominal plant power in kW *)
		MesFreqnom								: REAL;					(* (Hz) Defined nominal plant freq in Hz *)
		MesUnom									: REAL;					(* (V)  Defined nominal plant voltage in V *)
		MesNbINV								: UINT;					(* (NA) Number OF inverters installed on site *) 

		MesCPWrite								: BOOL;					(* (NA) 0: PPC not sending frames to inverters. 1: PPC sending frames to inverters *)
		MesState_QDistribAlgo					: BOOL;					(* (NA) activate Q distribution algorithm. 0: disable. 1: enable *)
		
// Inverter Status Words

		MesInvStatus							: ARRAY[1..11] OF WORD;	(* (NA) Status Words of Inverters *)

END_STRUCT	
END_TYPE

// ---- 01_Equipement_Library/ProtectRelay/ProtectRelay_Micom.TcDUT
///////////
// Structure For I35. Main Operating Data to be saved ( ex: OPC ) .  
//////////
TYPE ProtectRelay_Micom :
STRUCT
	
		MesData						: ProtectRelay;			(*	(NA) Protection relay									    *)
                                                        	                                               
		                                    				                                                             
		MesU						: REAL;					(* (V) Average Phase to Phase Voltage                           *)
	                                                    	
		MesV1						: REAL ;        		(* (V) Average Phase to Phase Voltage                           *)
		MesV2						: REAL ;				(* (V) Average Phase to Phase Voltage                           *)
		MesV3						: REAL ;				(* (V) Average Phase to Phase Voltage                           *)
		MesV0						: REAL ;				(*(V) Measured  maximal residual Voltage           			    *)
       			                                        	                   
		MesP						: REAL; 				(* (Kw)Power on Grid                                            *)
		MesQ						: REAL;					(* (kvar) Power on grid                                         *)
		MesS						: REAL;					(* (KVA) Power apparent                                         *)
		MesCosPhi					: REAL;					(* (NA) power factor                                            *)
		MesTanPhi					: REAL; 				(* (NA) Cal : tan Phi                                           *)
		   

                                 			                                                        
		MesStopPP_UminLong			: BOOL; 				(* (NA) PP is stopping during 2min, because of Long GTE fault	*)
		MesHomopol_Def				: BOOL;                 (* (NA)  Homopolar power default*)                   			                                                          

		EActProd					: REAL; 				(* (MWh) Active Energy Produced                                 *)
		EActCons					: REAL; 				(* (MWh) Active Energy Consummed                                *)
		EReactProd					: REAL; 				(* (MVArh) Reactive Energy Produced                             *)
		EReactCons					: REAL; 				(* (MVArh) Reactive Energy Consummed                            *)
		                                    			                                                           
	// Relais Input                         			
		Input11						: BOOL;					(* (NA) Input 11 du relais de protection                        *)
		Input12                     : BOOL;					(* (NA) Input 12 du relais de protection                        *)
		Input13                     : BOOL;					(* (NA) Input 13 du relais de protection                        *)
		Input14                     : BOOL;					(* (NA) Input 14 du relais de protection                        *)
		Input21						: BOOL;					(* (NA) Input 21 du relais de protection                        *)
		Input22						: BOOL;					(* (NA) Input 22 du relais de protection                        *)
		Input23						: BOOL;					(* (NA) Input 23 du relais de protection                        *)
		Input24						: BOOL;					(* (NA) Input 24 du relais de protection                        *)
		Input25						: BOOL;					(* (NA) Input 25 du relais de protection                        *)
		Input26						: BOOL;					(* (NA) Input 26 du relais de protection                        *)
		
				
END_STRUCT
END_TYPE

// ---- 01_Equipement_Library/ProtectRelay/ProtectRelay_SchP30U30.TcDUT
///////////
// Structure for Schneider P30U30. Main Operating Data to be saved (ex: OPC).  
//////////
TYPE ProtectRelay_SchP30U30:
STRUCT

		MesData						: ProtectRelay;		(*	(NA) Protection relay									    *)                                                                                                     
		                                    			                                                             
		MesU						: REAL;				(* (V) Average Phase to Phase Voltage                           *)
		MesV1						: REAL;        		(* (V) Average Phase to Phase Voltage                           *)
		MesV2						: REAL;				(* (V) Average Phase to Phase Voltage                           *)
		MesV3						: REAL;				(* (V) Average Phase to Phase Voltage                           *)
       	MesV0						: REAL;				(* (%) Residual voltage				                            *)
       			                                                           
		MesP						: REAL; 			(* (Kw)Power on Grid                                            *)
		MesQ						: REAL;				(* (kvar) Power on grid                                         *)
		MesS						: REAL;				(* (KVA) Power apparent                                         *)
		MesCosPhi					: REAL;				(* (NA) Power factor                                            *)
		MesTanPhi					: REAL; 			(* (NA) Tan Phi                                                 *)		                                    			                                                       

	// Energy		                                    			                                                          
		E_P_Prod					: REAL; 			(* (MWh) Active Energy Produced                                 *)
		E_P_Cons					: REAL; 			(* (MWh) Active Energy Consummed                                *)
		E_Q_Prod					: REAL; 			(* (MVArh) Reactive Energy Produced                             *)
		E_Q_Cons					: REAL; 			(* (MVArh) Reactive Energy Consummed                            *)
	
	// Positions
		MesInterr_Opened			: BOOL;				(* (NA) Interruptor opened*)
		MesSect_Opened				: BOOL;				(* (NA) Interruptor opened*)
		MesEartch_Opened			: BOOL;				(* (NA) Earthing switch opened*)
		MesSpring_Charged			: BOOL;				(* (NA) Spring  charged*)
		MesComutLocal				: BOOL; 			(* (NA) Selector state local/remote. 0 = remote, 1 = local		*)
		MesCtoDisparo_Opened		: BOOL;				(* (NA) cto disparo opened*)
		                                    			                                                           
	// Relais Input                         			                                                              
		Input11						: BOOL;				(* (NA) Input 11 du relais de protection                        *)
		Input12                     : BOOL;				(* (NA) Input 12 du relais de protection                        *)
		Input13                     : BOOL;				(* (NA) Input 13 du relais de protection                        *)
		Input14                     : BOOL;				(* (NA) Input 14 du relais de protection                        *)
		Input21						: BOOL;				(* (NA) Input 21 du relais de protection                        *)
		Input22						: BOOL;				(* (NA) Input 22 du relais de protection                        *)
		Input23						: BOOL;				(* (NA) Input 23 du relais de protection                        *)
		Input24						: BOOL;				(* (NA) Input 24 du relais de protection                        *)
		Input25						: BOOL;				(* (NA) Input 25 du relais de protection                        *)
		Input26						: BOOL;				(* (NA) Input 26 du relais de protection                        *)
		
	// Trip / alarms
		MesAlarmImax				: BOOL; 		 	(* (NA) Imax alarm 50/51 										*)
		MesAlarmImin				: BOOL; 		 	(* (NA) Imin alarm 37									  		*)		
		MesAlarmUmin				: BOOL;		 		(* (NA) Umin alarm 27											*)
		MesAlarmUmax				: BOOL;		 		(* (NA) Umax alarm 59											*)		
		MesAlarmFmax				: BOOL;		 		(* (NA) Fmax and Fmin alarm fX81								*)
		MesAlarmFmin				: BOOL;		 		(* (NA) Fmin alarm 81U											*)
		
		MesPPStop_Lgte				: BOOL; 			(* (NA) PP is stopping during 2min, because of a long GTE fault	*)
		
END_STRUCT
END_TYPE

// ---- 01_Equipement_Library/ProtectRelay/ProtectRelay_Siprotec.TcDUT
TYPE ProtectRelay_Siprotec :
STRUCT
	
	MesData					: ProtectRelay;
	
	MesComutLocal			: BOOL;	(**)
	MesTCSAlarm				: BOOL; (* Alarme TCS (Supervision circuit de déclenchement) *)
	MesVrAnomaly			: BOOL; (* Anomalie VR (tension résiduelle) *)
	MesTripSynthesis		: BOOL; (* Trip Synthesis *)
	
	// 3X Variables                 
	
	MesI					: REAL; (* (A) Current phase average *)                                
	MesI1					: REAL; (* (A) Current phase 1*)
	MesI2					: REAL; (* (A) Current phase 2*)
	MesI3					: REAL; (* (A) Current phase 3*)
	MesIn					: REAL; (* (A) Current phase n*)
	MesV1					: REAL; (* (V) Voltage phase 1*)
	MesV2					: REAL; (* (V) Voltage phase 2*)
	MesV3					: REAL; (* (V) Voltage phase 3*)
	MesU12					: REAL; (* (V) Voltage phase 12*)
	MesU23					: REAL; (* (V) Voltage phase 23*)
	MesU31					: REAL; (* (V) Voltage phase 31*)
	MesUn					: REAL; (* (V) Voltage phase n*)
	MesP					: REAL; (* (kW) Active Power calculated (from current, power and cosphi because otherwise not precise)*)
	MesQ					: REAL; (* (kVAr) Reactive Power *)
	MesS					: REAL; (* (kVA) Apparent Power*)
	MesFreq					: REAL; (* (Hz) Frequency*)
	MesCosPhi				: REAL; (* (NA) CosPhi*)
	
END_STRUCT
END_TYPE

// ---- 01_Equipement_Library/ProtectRelay/ProtectRelay_SMNS7L86.TcDUT
///////////
// Structure Siemens 7UT85 protection relay.  
//////////
TYPE ProtectRelay_SMNS7L86 :
STRUCT
	
		MesData					: ProtectRelay;		(* (NA) Protection relay								 			*)
        MesLiveContact			: BOOL;				(* (NA)*)																		
        MesAuxTrip				: BOOL;				(* (NA)*)                                                                       
        MesTripVT12				: BOOL;				(* (NA)*)                                                                       
        MesTripVT3				: BOOL;				(* (NA)*)                                                                       
        MesAlarmTripCircuit1	: BOOL;				(* (NA)*)                                                                       
        MesAlarmTripCircuit2	: BOOL;				(* (NA)*)                                                                       
		MesLocalMode			: BOOL;				(* (NA) Cell in local mode. 0=Remote, 1=Local						*)          
		MesRemoteMode			: BOOL;				(* (NA) Cell in local mode. 0=Local, 1=Remote						*)          
		MesOpened_52 			: BOOL;				(* (NA) SWITCH 52-2 OPEN. 0=Close, 1=Open   						*)          
		MesClosed_52			: BOOL;				(* (NA) SWITCH 52-2 CLOSED. 0=Open 1=Closed  						*)          
		MesOpened_89     		: BOOL;				(* (NA) PAT 89T-2 SWITCH OPEN. 0=close, 1=Open   					*)          
		MesClosed_89  			: BOOL;				(* (NA) PAT 89T-2 SWITCH CLOSED. 0=open, 1=Close		       		*)          
		MesOpened_89T     		: BOOL;				(* (NA) PAT 89T-2 SWITCH OPEN. 0=close, 1=Open   					*)          
		MesClosed_89T  			: BOOL;				(* (NA) PAT 89T-2 SWITCH CLOSED. 0=open, 1=Close		       		*)          
		MesAlarmSF6Pressure     : BOOL;             (* (NA)SF6 Pressure                                                 *)          
		MesGeneralTrip_TSA      : BOOL;             (* (NA)General Trip a TSA                                           *)          
		MesTrip_ANSI_86         : BOOL;             (* (NA)ANSI 86 Trip                                                 *)          
		MesTrip_ANSI_5051       : BOOL;             (* (NA)ANSI 50/51 Trip                                              *)          
		MesTrip_ANSI_50n51n     : BOOL;             (* (NA)ANSI 50N/51N Trip                                            *)          
		MesTrip_ANSI_50BF		: BOOL;				(* (NA) ANSI 50BF Trip : Breaker Failure							*)
		MesTrip_ANSI_87L        : BOOL;             (* (NA)ANSI 87L Trip                                                *)          
		MesTrip_ANSI_59         : BOOL;             (* (NA)ANSI 59 Trip                                                 *)          
		MesTrip_ANSI_59n        : BOOL;             (* (NA)ANSI 59N Trip                                                *)          
		MesTrip_ANSI_27         : BOOL;             (* (NA)ANSI 27 Trip                                                 *)          
		MesTrip_ANSI_81U        : BOOL;             (* (NA)ANSI 81U                                                     *)  		
		MesTrip_ANSI_81O        : BOOL;             (* (NA)ANSI 81O                                                     *)  		
		
		
		MesVTrip52_2 			: BOOL;				(* CHANGE IT (NA) TRIGGER CIRCUIT VOLTAGE 1 52-2. 0=Alarm 1=Normal 	*)
		MesTrip52_2 			: BOOL;				(* CHANGE IT(NA) TRIGGER CIRCUIT 1 52-2 OK WIRED 0=Alarm 1=Normal 	*)

		MesAlarmInterlocking	: BOOL;				(* (NA) interlocking alarm*)
		MesSpring_Loaded		: BOOL;				(* (NA) loaded spring*)

		                    	
		MesAlarmImaxN			: BOOL; 			(* (NA) Imax neutral alarm, ANSI Trip 50N, 51N synthesis			*)
		MesAlarmGas				: BOOL;				(* (NA) Cell gas pressure is low. 0=Normal 1=Alarm  		        *)                                      	
    	MesAlarmPower	  		: BOOL;				(* (NA) Power failure alarm 		    							*)
		MesAlarmAbnormal  		: BOOL;				(* (NA) Alarm for abnormal functionning 							*)
                            	  	                                               	                                    			                                                           
		MesV1					: REAL;				(* (V) Voltage of phase 1											*)
		MesV2					: REAL;				(* (V) Voltage of phase 2											*)
		MesV3					: REAL;				(* (V) Voltage of phase 3											*)
                            	
		MesIn					: REAL; 			(* (A) Current phase n*)
		MesUn					: REAL; 			(* (V) Voltage phase n												*)
		MesP					: REAL; 			(* (kW) Active Power calculated (from current, power and cosphi because otherwise not precise)*)
		MesQ					: REAL; 			(* (kVAr) Reactive Power *)
		MesS					: REAL; 			(* (kVA) Apparent Power*)
		MesCosPhi				: REAL; 			(* (NA) CosPhi*)

		OUT_CmdOpen				: BOOL;				(* (NA) Cmd To open CB*)
		OUT_CmdClose			: BOOL;				(* (NA) Cmd To close CB*)
		
END_STRUCT
END_TYPE

// ---- 01_Equipement_Library/ProtectRelay/ProtectRelay_Standard.TcDUT
///////////
// Structure For I35. Main Operating Data to be saved (ex: OPC).  
//////////
TYPE ProtectRelay_Standard :
STRUCT
	MesData			: ProtectRelay ; 
		
END_STRUCT
END_TYPE

// ---- 01_Equipement_Library/ProtectRelay/ProtectRelay_Flair23DM.TcDUT
TYPE ProtectRelay_Flair23DM :
STRUCT
		MesData						: ProtectRelay;		(* (NA) Protection relay			  *)
               
		MesV1						: REAL ; 			(* (V) Output Phase Voltage Phase 1   *)
		MesV2						: REAL ; 			(* (V) Output Phase Voltage Phase 2   *)
		MesV3						: REAL ; 			(* (V) Output Phase Voltage Phase 3   *)
		MesV0						: REAL ; 		    (* (V) Residual Voltage				  *)
		
		MesStateCom					: BOOL ; 			(* (NA) False=NotOK. Device did not respond successfully to most recent read/write request. True= Device is responding normally *)
	  	
		ControlWord					: WORD ; 			(* (NA) Control Word				 *)
	   	StatusWord					: WORD ; 			(* (NA) Status Word                  *)
		CalToggleWrite				: BOOL ;			(* (NA) True := read authorised      *)
		CalToggleRead				: BOOL ;			(* (NA) True := Write authorised     *)
		       
END_STRUCT
END_TYPE

// ---- 01_Equipement_Library/ProtectRelay/ProtectRelay_NSXCB.TcDUT
TYPE ProtectRelay_NSXCB :
STRUCT
		MesData						: ProtectRelay;			(* (NA) Protection relay				*)
               
		MesStatCom					: BOOL; 				(* (NA) False:=.:NotOK.Device did notrespond successfullyto most recentread orwrite request, TRUE := Device is responding normally *)
	                                        				
		MesMaxFreq					: REAL; 				(* (Hz) Frequence max					*)
		                                    				
		MesP1						: REAL; 				(* (kW) Active poweron phase 1 (P1) 	*)
		MesP2						: REAL; 				(* (kW) Active poweron phase 2 (P1) 	*)
		MesP3						: REAL; 				(* (kW) Active poweron phase 3 (P1) 	*)
        MesPtot						: REAL; 				(* (kW) Total active power(Ptot)    	*)
		                                    				
		MesQ1						: REAL; 				(* (kvar) Reactive poweron phase 1 (Q1) *)
		MesQ2						: REAL; 				(* (kvar) Reactive poweron phase 1 (Q2) *)
		MesQ3						: REAL; 				(* (kvar) Reactive poweron phase 1 (Q3) *)
		MesQtot						: REAL; 				(* (kvar) Total reactive power(Qtot)    *)
		                                    				
		MesS1						: REAL; 				(* (kVA) Apparent power on phase 1 		*)
		MesS2						: REAL; 				(* (kVA) Apparent power on phase 2 		*)
		MesS3						: REAL; 				(* (kVA) Apparent power on phase 3 		*)
		MesStot						: REAL;					(* (kVA) Total apparentpower(Stot) 		*)
		                                    				
		MesEAct						: REAL; 				(* (Wh)  Active energy       			*)
		MesEReact					: REAL; 				(* (VArh)Reactive energy		   		*)
		                                    				
		MesCosPhi1					: REAL; 				(* (pu) Power factor on phase 1  		*)
		MesCosPhi2					: REAL; 				(* (pu) Power factor on phase 2  		*) 	
		MesCosPhi3					: REAL; 				(* (pu) Power factor on phase 3  		*)
		MesCosPhi					: REAL; 				(* (pu) Power factor on phase Tot		*)
		
		MesToggleWrite				: BOOL;					(* (NA) Cal: True := read authorised 	*)
		MesToggleRead				: BOOL;					(* (NA) Cal: True := Write authorised	*)
		                                    	                                                	
		
		
		
		
		
		
END_STRUCT
END_TYPE

// ---- 01_Equipement_Library/ProtectRelay/ProtectRelay_PACE100ST.TcDUT
TYPE ProtectRelay_PACE100ST :
STRUCT   
	
		Thermal_Overload			: REAL ; (* %  0 TO 250                         *)
	//Status                                 (*                                     *)
		Comut						: BOOL ; (* Cell's selector is in remote position    *)
		CB_Close					: BOOL ; (*  Cell is closes                                   *)
		CB_In_Alarm					: BOOL ; (*Cell is in alarm                                     *)
		Trip_Counter				: INT;   (*  Number of trip *)

                                  
		Mesdata 					: ProtectRelay;   (*                                     *)
        
END_STRUCT
END_TYPE

// ---- 01_Equipement_Library/ProtectRelay/ProtectRelay_REFIO.TcDUT
TYPE ProtectRelay_REFIO :
STRUCT
	
	MesData				: ProtectRelay ; 	(* Object 								    *)
	MesTransfoAlarm		: BOOL ; 	(* Transfo alarm                              *)
	MesSWOpened			: BOOL ;	(* Sectionneur de ligne ouvert              *)
	MesSWClosed			: BOOL ; 	(* Sectionneur de ligne fermé               *)
	MesEarth			: BOOL ; 	(* Earthing                                 *)
	MesSF6Low			: BOOL ; 	(* SF6 gaz is low                           *)
	MesSF6Unsufficient	: BOOL ; 	(* Sf6  is unsufficient                     *)
	MesTransfoWarning	: BOOL ; 	(* Transfo warning                            *)
	MesOpened			: BOOL ; 	(* Disjoncteur opened                       *)
	MesClosed			: BOOL ; 	(* Disjoncteur is closed                    *)
	MesComutLocal		: BOOL ; 	(* Commutateur Local/Distant.               *)
	
	
END_STRUCT
END_TYPE

// ---- 01_Equipement_Library/ProtectRelay/ProtectRelay.TcDUT
///////////
// Structure For I35. Main Operating Data to be saved (ex: OPC).  
//////////
TYPE ProtectRelay :
STRUCT
		MesI1						: REAL ; 			(* (A) Maximal Current measured before fault on phase 1*)
		MesI2						: REAL ;			(* (A) Maximal Current measured before fault on phase 2*)
		MesI3						: REAL ;			(* (A) Maximal Current measured before fault on phase 3*)
		MesI0						: REAL ; 			(*(A) Measured  maximal residual current               *)
		MesI						: REAL ;			(*(A) Phase current value (averaged)               	   *)
		                                        		                                                    
		MesFreq						: REAL ;			(* (Hz) Frequency measured                             *)
		                                        		                                                    
		MesImax1					: REAL ; 			(* (A) AC Max current during Fault phase 1             *)
		MesImax2                    : REAL ; 			(* (A) AC Max current during Fault phase 2             *)
		MesImax3                    : REAL ; 			(* (A) AC Max current during Fault phase 3		       *)
		MesImax0                    : REAL ; 			(* (A) AC Max residual current during Fault	           *)
		
		MesTripped                  : BOOL ;            (* Trip Synthesis *)                                        		                                                    
		MesAlarmCom					: BOOL ;			(* Communication Error with Sepam                      *)
                                                		                                                   
		MesAlarmTCS					: BOOL ; 			(* TCS in fault. RPN can not trip anymore              *)
		MesAlarmImax				: BOOL ; 			(* Imax alarm, ANSI Trip 50, 51 , 50G, 51G Synthesis                                       *)
		MesAlarmUmin				: BOOL ;			(* Short GTE Fault                                     *)
		MesAlarmUmin_Long			: BOOL ;			(* Long GTE FAULT                                      *)
      	MesAlarm_GTE3Time			: BOOL ; ;			(* 3 GTE FAULT   in 30 minutes                                   *)
		MesU12                      : REAL ;            (* (V) Voltage between phase 2 and phase 1 *)
		MesU23                      : REAL ;            (* (V) Voltage between phase 3 and phase 2 *)     
		MesU31                      : REAL ;            (* (V) Voltage between phase 1 and phase 3 *)                                                                                              
		
		MesWatchdog	                : BOOL ;            (* Watchdog *) 

		MesCP_Read					: BOOL := TRUE;	(* Cal Read function enable                            *)
		MesCP_Write					: BOOL := FALSE;	(* Cal Write function enable                           *)
		                                                                                                     
		MesAlarmCode				: WORD ; 			(* (NA) Internal Akuo AlarmCode                        *)
		MesWarningCode				: WORD ; 			(* (NA) Internal Akuo WarningCode                      *)
		MesEventCode				: WORD ; 			(* (NA) Internal Akuo EventCode		                   *)
		
END_STRUCT
END_TYPE

// ---- 01_Equipement_Library/ProtectRelay/ProtectRelay_S42.TcDUT
TYPE ProtectRelay_S42 :
STRUCT
	
	MesData							: ProtectRelay ; 	(* Object *)

	MesAlarm_Phase1					: BOOL ;(* Default Phase 1*)		
	MesAlarm_Phase2				    : BOOL ;(*Default Phase 2*)
	MesAlarm_Phase3				    : BOOL ;(*Default Phase 3*)
	MesAlarm_PhaseRpt			    : BOOL ;(*Default Phase RPT (relai presence tension ? ) *)
	MesAlarm_Ground				    : BOOL ;(*Default Ground*)
	MesAlarm_GroundRpt			    : BOOL ;(*Default Ground RPT (relai presence tension ? )*)
	MesAlarm_MaxUInverse			: BOOL ;(*Default Max UI Inverse*)
	MesAlarm_MaxP				    : BOOL ;(*Default Max P *)
	MesAlarm_CB		   			 	: BOOL ;(*Default Circuit breaker *)
	MesAlarm_Watchdog				: BOOL ;(* Défault watchdog*)						
	OUT_CmdOpen	   			 		: BOOL ;(* Circuit breaker Open Command*)
	OUT_CmdClose	    			: BOOL ;(*Circuit breaker Close Command*) 
                      
	MesU0					    	: REAL ;(*(V) Residual Voltage*)
	MesP							: REAL ;(*(kW) Active Power*)
	MesQ							: REAL ;(*(kVAr) Reactive Power*)
	MesCosPhi						: REAL ;(*(p.u) CospPhi*)
	
	MesAlarm_CablesOvercharge 		: BOOL; (*Cables Overcharge*) 		
    MesAlarm_FaultFrom225kV			: BOOL; (*Fault From 225 kV*)		
	
	
END_STRUCT
END_TYPE

// ---- 01_Equipement_Library/ProtectRelay/ProtectRelay_S48.TcDUT
///////////
// Structure For I35. Main Operating Data to be saved ( ex: OPC ) .  
//////////
TYPE ProtectRelay_S48 :
STRUCT
	
		MesData						: ProtectRelay;			(*	(NA) Protection relay									    *)
                                                        	                                               
		                                    				                                                             
		MesU						: REAL;					(* (V) Average Phase to Phase Voltage                           *)
	                                                    	
		MesV1						: REAL ;        		(* (V) Average Phase to Phase Voltage                           *)
		MesV2						: REAL ;				(* (V) Average Phase to Phase Voltage                           *)
		MesV3						: REAL ;				(* (V) Average Phase to Phase Voltage                           *)
       			                                        	                   
		MesP						: REAL; 				(* (Kw)Power on Grid                                            *)
		MesQ						: REAL;					(* (kvar) Power on grid                                         *)
		MesS						: REAL;					(* (KVA) Power apparent                                         *)
		MesCosPhi					: REAL;					(* (NA) power factor                                            *)
		MesTanPhi					: REAL; 				(* (NA) Cal : tan Phi                                           *)
		                                    			                                                          
		EActProd					: REAL; 				(* (MWh) Active Energy Produced                                 *)
		EActCons					: REAL; 				(* (MWh) Active Energy Consummed                                *)
		EReactProd					: REAL; 				(* (MVArh) Reactive Energy Produced                             *)
		EReactCons					: REAL; 				(* (MVArh) Reactive Energy Consummed                            *)
      		                                    			                                                           
	// Relais Input                         			

		Input11						: BOOL;					(* (NA) Input 11 du relais de protection                        *)
		Input12                     : BOOL;					(* (NA) Input 12 du relais de protection                        *)
		Input13                     : BOOL;					(* (NA) Input 13 du relais de protection                        *)
		Input14                     : BOOL;					(* (NA) Input 14 du relais de protection                        *)
		Input21						: BOOL;					(* (NA) Input 21 du relais de protection                        *)
		Input22						: BOOL;					(* (NA) Input 22 du relais de protection                        *)
		Input23						: BOOL;					(* (NA) Input 23 du relais de protection                        *)
		Input24						: BOOL;					(* (NA) Input 24 du relais de protection                        *)
		Input25						: BOOL;					(* (NA) Input 25 du relais de protection                        *)
		Input26						: BOOL;					(* (NA) Input 26 du relais de protection                        *)		
		


END_STRUCT
END_TYPE

// ---- 01_Equipement_Library/ProtectRelay/ProtectRelay_T20.TcDUT
///////////
// Structure For I35. Main Operating Data to be saved ( ex: OPC ) .  
//////////
TYPE ProtectRelay_T20 :
STRUCT
	// I35 Data measures
	
		MesData						: ProtectRelay; (*							*)							
                                           			(*                          *)
	                                       			(*                          *)
		MesFreq						: REAL;			(* (Hz) Frequence of grid   *)
		MesP						: REAL;			(* (Kw)Power on Grid        *)
		MesQ						: REAL;			(* (kvar) Power on grid     *)
		MesS						: REAL;			(* (KVA) Power apparent     *)
		                                   			(*                          *)
		MesTripProtec				: REAL;			(* A                        *)
		MesGlobalWarming		    : REAL;			(* % Au warming of TR       *)


END_STRUCT
END_TYPE

// ---- 01_Equipement_Library/ProtectRelay/ProtectRelay_T87.TcDUT
TYPE ProtectRelay_T87 :
STRUCT
	
	MesData							: ProtectRelay ; 		(* Object 								    *)

	MesAlarm_DiscordSectLigneHTB	: BOOL;   				(*DiscordSectLigneHTB*)
	MesAlarm_DiscordSectMaltHTB		: BOOL;   				(*DiscordSectMaltHTB	*)
	MesAlarm_DiscordSectDisjHTB		: BOOL;   				(*DiscordSectDisjHTB	*)
	MesAlarm_TeleCondamne			: BOOL;   				(*TeleCondamne		*)
	MesAlarm_DeTeleCondamne			: BOOL;   				(*DeTeleCondamne		*)
	MesAlarm_DiscordTeleCondamne	: BOOL;	  				(*DiscordTeleCondamne*)
                                                			
	MesAlarm_IoMaxCoteProd			: BOOL;   				(*IoMaxCoteProd*)
	MesAlarmUMax					: BOOL;   				(*UMax		*)
	MesAlarmUMax_Long				: BOOL;   				(*UMax_Long	*)
	MesAlarm_PhaseRpt				: BOOL;					(*PhaseRpt*)
	MesWarning_ImgTherm				: BOOL;					(*ImgTherm alarm*)
	MesAlarm_ImgTherm				: BOOL;					(*ImgTherm warning*)
	MesAlarm_DifferTransfo			: BOOL;					(*DifferTransfo*)
	MesAlarm_FreqMax				: BOOL;					(*FreqMax*)
	MesAlarm_FreqMin				: BOOL;					(*FreqMin*)	
	                                            			
	MesU0							: REAL;					(*(V) Residual Voltage*)
	MesP							: REAL;					(*(kW) Active Power*)	
	MesQ							: REAL;					(*(kVAr) Reactive Power*)
	

	
END_STRUCT
END_TYPE

// ---- 01_Equipement_Library/ProtectRelay/ProtectRelay_VIP410.TcDUT
TYPE ProtectRelay_VIP410 :
STRUCT
		MesData						: ProtectRelay; 	(* (NA) MesData 																												*)
		MesStatCom					: BOOL ; 			(* (NA) False: device did not respond successfully to most recent read or write request, True: device is responding normally	*)
		MesAvgI1					: REAL ; 			(* (A) Phase 1 Average current                                                                                       			*)
		MesAvgI2					: REAL ; 			(* (A) Phase 2 Average current                                                                                       			*)
		MesAvgI3					: REAL ; 			(* (A) Phase 3 Average current                                                                                       			*)
		MesI0Fault					: REAL ; 			(* (A) Fault current                                                                                                 			*)
		StatusWord					: WORD ; 			(* (NA) Status Word                                                                                                     		*)
		ControlWord					: WORD ; 			(* (NA) Control Word                                                                                                    		*)
END_STRUCT
END_TYPE

// ---- 01_Equipement_Library/ProtectRelay/ProtectRelay_WIP1.TcDUT
///////////
// Structure For I35. Main Operating Data to be saved ( ex: OPC ) .  
//////////
TYPE ProtectRelay_WIP1 :
STRUCT
	// I35 Data measures
	MesData					: ProtectRelay ; (**)


	
END_STRUCT
END_TYPE

// ---- 01_Equipement_Library/Router/Router.TcDUT
TYPE Router :
STRUCT
		MesWatchdog	        : BOOL ; 	(* Watchdog*)
		
		MesAlarmCode		: WORD ;	(* (NA) Internal Akuo AlarmCode		*)
		MesWarningCode		: WORD ; 	(* (NA) Internal Akuo WarningCode   *)
		MesEventCode		: WORD ; 	(* (NA) Internal Akuo EventCode	    *)
		
END_STRUCT
END_TYPE

// ---- 01_Equipement_Library/Router/Router_Standard.TcDUT
TYPE Router_Standard :
STRUCT
		MesData				: Router ;  (* Object *)

		
END_STRUCT
END_TYPE

// ---- 01_Equipement_Library/Sensors/ANA/ANA.TcDUT
TYPE ANA :
STRUCT
	Value 					: REAL ;	(* (-) Analogic Value 					*)
	                                    
	MesAlarmCode			: WORD ;	(* (NA) Internal Akuo AlarmCode     *)
	MesWarningCode			: WORD ;    (* (NA) Internal Akuo WarningCode   *)
	MesEventCode			: WORD ;    (* (NA) Internal Akuo EventCode		*)

	MesCP_Read				: BOOL := TRUE;		(* (NA) CP for read purposes*)
END_STRUCT
END_TYPE

// ---- 01_Equipement_Library/Sensors/ANA/ANA_DevStd_Prom.TcDUT
TYPE ANA_DevStd_Prom :
STRUCT
	Value_Mean				: REAL ;	(* (-) Analogic mean value			*)
	Value_Devstd			: REAL ;	(* (-) Standard deviation value		*)
	
	MesAlarmCode			: WORD ;	(* (NA) Internal Akuo AlarmCode     *)
	MesWarningCode			: WORD ;    (* (NA) Internal Akuo WarningCode   *)
	MesEventCode			: WORD ;    (* (NA) Internal Akuo EventCode		*)

END_STRUCT
END_TYPE

// ---- 01_Equipement_Library/Sensors/ANA/ANA_DustIQ.TcDUT
TYPE ANA_DustIQ :
STRUCT
	Value_Mean				: REAL ;	(* (-) Analogic mean value							*)
	Value_Devstd			: REAL ;	(* (-) Standard deviation value						*)
	Value_Soiling			: REAL ; 	(* (-) To be changed 								*)
	
	MesAlarmCode			: WORD ;	(* (NA) Internal Akuo AlarmCode     				*)
	MesWarningCode			: WORD ;    (* (NA) Internal Akuo WarningCode   				*)
	MesEventCode			: WORD ;    (* (NA) Internal Akuo EventCode						*)

END_STRUCT
END_TYPE

// ---- 01_Equipement_Library/Sensors/ANA/ANA_Standard.TcDUT
TYPE ANA_Standard :
STRUCT
	
	MesData		: ANA; (* (NA) Child struct *)
END_STRUCT
END_TYPE

// ---- 01_Equipement_Library/Sensors/COM/AllInOne.TcDUT
TYPE AllInOne :
STRUCT
	
	MesWindSp 			: REAL ;		(* (m/s)	 Wind speed measurement of the weather station												        *)
	MesWindDir 			: REAL ;		(* (°) 		 Wind direction measurement of the weather station                                                  *)
	MesHygro			: REAL ;		(* (%) 		 Humidity measurement of the weather station                                                        *)
	MesTemp_Amb 		: REAL ;		(* (°C)		 Ambiant temperature measurement of the weather station                                             *)
	MesDewPoint			: REAL ;		(* (%) 		 Dew point measure of weather station                                                               *)
	MesRain1			: REAL ;		(* (count/h) Rain rate                                                                                          *)
	MesRain2			: REAL ;		(* (count/h) Rain rate                                                                                          *)
	MesRain3			: REAL ;		(* (count/h) Rain rate                                                                                          *)
                                       
	MesAlarmWindSp		: REAL ;		(* (NA) Alarm for the Wind speed : 0=OFF, 1 = Lower threshold, 2 = Higher threshold                                  *)
	MesAlarmWindDir		: REAL ;		(* (NA) Alarm for the Wind direction : 0=OFF, 1 = Lower threshold, 2 = Higher threshold                              *)
	MesAlarmTemp		: REAL ;		(* (NA) Alarm for the temp sensor : 0=OFF, 1 = Lower threshold, 2 = Higher threshold                                 *)
	MesAlarmHygro		: REAL ;		(* (NA) Alarm for the humidity sensor : 0=OFF, 1 = Lower threshold, 2 = Higher threshold                             *)
	MesAlarmDewPt		: REAL ;		(* (NA) Alarm for the dew point sensor : 0=OFF, 1 = Lower threshold, 2 = Higher threshold                            *)
	MesAlarmRain1		: REAL ;		(* (NA) Alarm for the rain sensor : 0=OFF, 1 = Lower threshold, 2 = Higher threshold                                 *)
	MesAlarmRain2		: REAL ;		(* (NA) Alarm for the rain sensor : 0=OFF, 1 = Lower threshold, 2 = Higher threshold                                 *)
	MesAlarmRain3		: REAL ;		(* (NA) Alarm for the rain sensor : 0=OFF, 1 = Lower threshold, 2 = Higher threshold                                 *)
	                                   
	MesAlarmCode		: WORD ;  	    (*  (NA) Alarm code Akuo    *)
	MesWarningCode		: WORD ;  	    (*  (NA) Warning code Akuo    *)
	MesEventCode		: WORD ; 	    (*  (NA) Event code Akuo    *)
	MesCP_Read			: BOOL := TRUE; (* (NA) Permanent condition for read *)
	
END_STRUCT
END_TYPE

// ---- 01_Equipement_Library/Sensors/COM/AllInOne_Standard.TcDUT
TYPE AllInOne_Standard :
STRUCT
	
	MesData			: AllInOne;
	
	MesPressure		: REAL; (*(bar) Pressure*)
	MesGHI			: REAL; (* (W/m²) Horizontal irradiance*)
	
	
END_STRUCT
END_TYPE

// ---- 01_Equipement_Library/Sensors/COM/DustIQ.TcDUT
TYPE DustIQ :
STRUCT
	MesSoilingRatio1				: REAL;  		(* (%) Soiling ratio measured by the DustIQ for sensor1 , in percentage (from 101% to 50%) after correction by transmission loss *)
	MesSoilingRatio2				: REAL;  		(* (%) Soiling ratio measured by the DustIQ for sensor2 , in percentage (from 101% to 50%) after correction by transmission loss *)
	                            	
	MesSoilingRatio					: REAL;  		(* (%) Soiling ratio measured by the DustIQ average of 2 sensors, in percentage (from 101% to 50%) after correction by transmission loss *)
	
	MesTemp_Panel					: REAL;			(* (°C) Panel temperature*)
	
	MesNeedForCalibration			: BOOL;			(* (NA) Informs need for calibration *)
	MesCalibrationDone				: BOOL;			(* (NA) Informs completion of calibration *)
	
	MesTiltDirection_X				: REAL;			(* (°) Tilt direction in long axis*)
	MesTiltDirection_Y				: REAL;			(* (°) Tilt direction in short axis*)
	
	MesAlarmCode					: WORD;			(* (NA) Akuo internal Alarm Code *)
	MesWarningCode					: WORD;         (* (NA) Akuo internal Warning Code *)
	MesAlarmCom						: BOOL;         (* (NA) Communication alarm*)
	MesCP_Read						: BOOL := TRUE;         (* (NA) Permanent condition for read *)
END_STRUCT
END_TYPE

// ---- 01_Equipement_Library/Sensors/COM/DustIQ_Standard.TcDUT
TYPE DustIQ_Standard :
STRUCT
	MesData : DustIQ ; (* Child struct  *)
END_STRUCT
END_TYPE

// ---- 01_Equipement_Library/Sensors/COM/PV_temp_sensor.TcDUT
TYPE PV_temp_sensor :
STRUCT
	
	MesData      : ANA;
	MesCP_Read	 : BOOL;	
	

END_STRUCT
END_TYPE

// ---- 01_Equipement_Library/Sensors/COM/SMP1X.TcDUT
TYPE SMP1X :
STRUCT
	MesData						: ANA; 			(**)

	
	MesIDAlarm					: WORD;			(**)
	MesCP_Read					: BOOL;			(**)

END_STRUCT
END_TYPE

// ---- 01_Equipement_Library/Sensors/TOR/TOR.TcDUT
TYPE TOR :
STRUCT
	
	MesAlarmState 		 		: BOOL  ;		(* TRUE = ALARM													*)
	MesCountAlarm				: UDINT ; 		(* Count the number of time the alarm has been triggered.       *)
                                                (*                                                              *)
	MesAlarmCode				: WORD ;		(* (NA) Internal Akuo AlarmCode                                 *)
	MesWarningCode				: WORD ;   	 	(* (NA) Internal Akuo WarningCode                               *)
	MesEventCode				: WORD ;	 	(* (NA) Internal Akuo EventCode		                            *)

END_STRUCT		
END_TYPE

// ---- 01_Equipement_Library/Sensors/TOR/TOR_CB.TcDUT
TYPE TOR_CB :
STRUCT
	
	MesData					: TOR ;		(* MesData 											 *)
	MesTripped				: BOOL;		(* (NA) CB is tripped*)
	MesCP_Open				: BOOL; 	(* (NA) Permanent condition to open CB *)
	MesCP_Close				: BOOL; 	(* (NA) Permanent condition to close CB *)
END_STRUCT		
END_TYPE

// ---- 01_Equipement_Library/Sensors/TOR/TOR_Standard.TcDUT
TYPE TOR_Standard :
STRUCT
	
	MesData					: TOR ;		(* MesData 											 *)

END_STRUCT		
END_TYPE

// ---- 01_Equipement_Library/Sensors/TOR/TOR_Rain.TcDUT
TYPE TOR_Rain :
STRUCT
	
	MesData					: TOR ;		(* MesData 											 *)
	MesRainFall_LastHour  	: REAL;   	(* (mm)Amount of water fall during the last hour	 *)
	MesRainFall_LastDay   	: REAL;   	(* (mm)Amount of water fall during the last Day (mm) *)
	MesRainFall_LastMonth 	: REAL;   	(* (mm)Amour of water fall during the last Year (mm) *)
	                           
	AvgmmHour	  			: REAL; 	(* (mm)Hourly AVG of water fall                      *)
	AvgmmDay   				: REAL;     (* (mm)Daily AVG of water fall                       *)
	AvgmmMonth 				: REAL;     (* (mm) Monthly AVG of water fall                    *)
	
END_STRUCT
END_TYPE

// ---- 01_Equipement_Library/TAC/TAC.TcDUT
TYPE TAC :
STRUCT
	
	MesFault				: BOOL;		(* (NA) Fault detected*)
	OUT_CmdActivated		: BOOL;		(* (NA) The TAC is ordered to be active*)
	MesActivated			: BOOL;		(* (NA) The TAC has been measured to be active*)
	MesCmdDisconnect		: BOOL;		(* (NA) TAC received a disonnect order from Grid Manager*)
	MesAlarmCode			: WORD;		(* (NA) Akuo Internal Alarm Code*)
	MesWarningCode			: WORD;		(* (NA) Akuo Internal Warning Code*)
END_STRUCT
END_TYPE

// ---- 01_Equipement_Library/TAC/TAC_Standard.TcDUT
TYPE TAC_Standard :
STRUCT
	MesData : TAC; 			(* Main Structure *)
END_STRUCT
END_TYPE

// ---- 01_Equipement_Library/Tariff Meter/EM_ION8650.TcDUT
TYPE EM_ION8650 :
STRUCT
	
	MesData					: EM; 			(* (NA) MesData							*)
	
	//MesAlarmPower		  	: BOOL;			(* (NA) Power failure alarm 		    *)
	MesAlarmAbnormal  		: BOOL; 		(* (NA) Alarm for abnormal functionning *)	
	MesLossPhase			: BOOL;			(* (NA) Loss of 1 or more TC phases		*)
	
END_STRUCT
END_TYPE

// ---- 01_Equipement_Library/Tariff Meter/EM_Standard.TcDUT
TYPE EM_Standard :
STRUCT
	
	MesData			: EM ; 

END_STRUCT
END_TYPE

// ---- 01_Equipement_Library/Tariff Meter/EM.TcDUT
TYPE EM :
STRUCT
	
	MesEActCons				: REAL ; 		(* Value of Active Energy consumed		*)
	MesEActProd				: REAL ;		(* Value of Active Energy produced      *)
	MesEReactCons			: REAL ;		(* Value of Reactive Energy consumed    *)
	MesEReactProd			: REAL ;		(* Value of Reactive Energy produced    *)
	                                                                             
	MesAlarmCode			: WORD ;	 	(* (NA) Internal Akuo AlarmCode         *)
	MesWarningCode			: WORD ; 		(* (NA) Internal Akuo WarningCode       *)
	MesEventCode			: WORD ; 		(* (NA) Internal Akuo EventCode	        *)

END_STRUCT
END_TYPE

// ---- 01_Equipement_Library/Tracker/NCU.TcDUT
TYPE NCU :
STRUCT
	// Data for Trackers aggregator
	

		MesAlarmCom			: BOOL ;
		
		MesAlarmCode		: WORD ;
		MesWarningCode 		: WORD ; 
		MesEventCode		: WORD ; 
		
		MesCP_Read			: BOOL := TRUE;
		MesCP_Write			: BOOL  ;
	
		
		
END_STRUCT
END_TYPE

// ---- 01_Equipement_Library/Tracker/NCU_Axial.TcDUT
TYPE NCU_Axial :
STRUCT
	// Data for Trackers aggregator
	
		MesData				: NCU ;
	
		AX_TRK			: ARRAY[1..CstNbTrk_NCU_G] OF TRK_Axial;
		
		MesRSUGlobal		: WORD ; 
	//	MesAnemoAlarm		: WORD ; 
		MesComNCUAlarm		: WORD ; 
		MesSnow				: REAL ; 
		MesWindSpeed		: REAL ; 
		MesWindDir			: REAL ; 
		
		MesForceWindCmd		: WORD ; 
		MesForceCleaningCmd	: WORD ; 
		MesForceSnowCmd		: WORD ; 
		

		MesWindAlarm		: BOOL ; 
		
		CalCPEmergency		: BOOL;
		CalCPWindPos		: BOOL;
		CalCPSnowPos		: BOOL;
		CalCPCleaningPos	: BOOL;
		
		
END_STRUCT
END_TYPE

// ---- 01_Equipement_Library/Tracker/TRK.TcDUT
TYPE TRK :
STRUCT
	// Structure for all tables with trackers
	
		MesAngle			: REAL ; 	// rad . -Pi , Pi . Tracker angle . 
		MesAngleTarget		: REAL ; 	// rad . -Pi .. pi . Tracker angle target 
	
	
END_STRUCT
END_TYPE

// ---- 01_Equipement_Library/Tracker/TRK_Axial.TcDUT
TYPE TRK_Axial :
STRUCT
	// Structure for all tables with trackers
		MesData				: TRK ; 
		MesImaxmotor		: REAL;		// A . Motor Maximal Current 
		MesImotor			: REAL;		// A . Motor Current
		MesStatusSynthesis	: WORD ; 
END_STRUCT
END_TYPE

// ---- 01_Equipement_Library/Transfo/TapChanger.TcDUT
TYPE TapChanger :		// Regleur Transfo 
STRUCT

	MesAlarm						: BOOL;          (* *)
	MesAlarm_Discordance			: BOOL;          (* *)
	MesAlarm_NoOutletDetected		: BOOL;          (* *)
	MesModeAuto						: BOOL;          (* *)
	MesModeManual					: BOOL;          (* *)
	MesState_ManoeuverAuthorized	: BOOL;	         (* *)
	OUT_CmdRampUp					: BOOL;          (* *)
	OUT_CmdRampDown					: BOOL;          (* *)
	       	
	MesIDPosPrise1to21 				: REAL;          (*PosPrise1to21 *)


END_STRUCT
END_TYPE

// ---- 01_Equipement_Library/Transfo/Transfo.TcDUT
TYPE Transfo :
STRUCT
	
    MesWarningTemp				: BOOL ;	(* Transfo Temperature Warning		    *)
    MesAlarmTemp				: BOOL ;	(* Transfo Temperature Alarm		    *)
    MesAlarmGas					: BOOL ;	(* Transfo Gas Alarm			        *)
    MesAlarmOilLevel			: BOOL ;	(* Transfo Oil Level Alarm		        *)
    MesAlarmsSynthesis			: BOOL ;	(* Transfo Synthesis Alarm              *)
	MesAlarmPowerSupply			: BOOL ;	(* Transfo Power Supply Alarm           *)
	MesAlarmPressure			: BOOL ;	(* Pressure Alarm          				*)
                                                                             
	MesAlarmCode				: WORD ;  	(* (NA) Internal Akuo AlarmCode         *)
	MesWarningCode				: WORD ; 	(* (NA) Internal Akuo WarningCode       *)
	MesEventCode				: WORD ; 	(* (NA) Internal Akuo EventCode	        *)

END_STRUCT
END_TYPE

// ---- 01_Equipement_Library/Transfo/Transfo_HV.TcDUT
TYPE Transfo_HV :
STRUCT

	MesData						: Transfo ; (* Transfo*)

	MesWarningGas					: BOOL  ; (* Buchholz warning*)

	MesWarning_TempLevel1			: BOOL  ; (*ImgTherm1erStade*)
	MesWarning_TempLevel2			: BOOL  ; (*ImgTherm2ndStade*)
	MesTrigger_Deletion				: BOOL  ; (*TransfoDcltSurpression*)

	MesTransfoRefrigLocal			: BOOL  ; (*TransfoRefrigLocal*)
	
	MesTrigger_NonReturnValve		: BOOL  ; (*declenchement clapet anti retour*)
	MesTrigger_ProtectRelay			: BOOL  ; (*DcltRelaisProtectRegl*)
	MesAlarm_TapChanger				: BOOL  ; (*Fault TapChanger*)
	
	


END_STRUCT
END_TYPE

// ---- 01_Equipement_Library/Transfo/Transfo_MV.TcDUT
TYPE Transfo_MV :
STRUCT
	
	MesData						: Transfo ; (* MesData *)


END_STRUCT
END_TYPE

// ---- 01_Equipement_Library/UPS/UPS_CXC.TcDUT
///////////
// Structure For I35. Main Operating Data to be saved ( ex: OPC ) .  
//////////
TYPE UPS_CXC :
STRUCT
	
	MesData				: UPS ; 	(* Object 									*)
	            		            (*                                          *)
	MesU				: REAL ; 	(*(V) AC voltage                            *)
	MesIload			: REAL ; 	(*(A) DC Load current                       *)
	MesUBatt			: REAL ; 	(*(V) Battery voltage                       *)
	MesIBatt			: REAL ; 	(*(A) Battery Current                       *)
	MesSoC  			: REAL ; 	(*(%) Battery SoC                           *)
	MesIdc  			: REAL ; 	(*(A) battery + load Current                *)

	
	MesOverTempBatt 	: BOOL ; 	(* OverTemperature of the battery alarm		*)
	MesCBUpsOpened		: BOOL ; 	(* UPS CB opened alarm                      *)
	
		
	
END_STRUCT
END_TYPE

// ---- 01_Equipement_Library/UPS/UPS.TcDUT
///////////
// Structure for UPS. Main Operating Data to be saved (ex: OPC)  
//////////
TYPE UPS :
STRUCT
		MesDischarging				: BOOL ; 			(* (NA) Battery is discharging		*)
		MesAlarm_Ulow				: BOOL ; 			(* (NA) Battery is almost empty     *)
		MesAlarmState				: BOOL ; 			(* (NA) Fault on the charger        *)
		MesUdc  					: REAL ; 			(* (V) DC Load voltage              *)
       		
		
		MesAlarmCode				: WORD ; 			(* Internal Akuo Alarm Code         *)
		MesWarningCode				: WORD ; 			(* Internal Akuo Warning Code       *)
		MesEventCode				: WORD ; 			(* Internal Akuo Warning Code 	    *)
        
		MesCP_Read					: BOOL := TRUE ;   (* Read function enable             *)
		MesAlarmCom					: BOOL ; 			(* Communication alarm              *)
	
END_STRUCT
END_TYPE

// ---- 01_Equipement_Library/UPS/UPS_Eneris.TcDUT
///////////
// Structure For I35. Main Operating Data to be saved (ex: OPC).  
//////////
TYPE UPS_Eneris :
STRUCT
	// I35 Data measures
		MesData                     : UPS;  (* MesData *)
		
END_STRUCT
END_TYPE

// ---- 01_Equipement_Library/UPS/UPS_MCSU4.TcDUT
///////////
// Structure For I35. Main Operating Data to be saved ( ex: OPC ) .  
//////////
TYPE UPS_MCSU4 :
STRUCT
	
	MesData				: UPS ; 	(* (NA) Object										*)
	            		                                                            	
	MesAlarmUmax		: BOOL; 	(* (NA) Over voltage alarm 							*)
                                                                                    	
	MesAlarmTemp		: BOOL; 	(* (NA) Ambient temperature high alarm 				*)
	MesAlarmTemp_Bat	: BOOL;		(* (NA) Battery temperature high alarm		    	*)
                                                                                    	
	MesAlarmI_diff		: BOOL;		(* (NA) Differential battery discharge current alarm*)
	MesAlarmI_Earth		: BOOL;		(* (NA) Earth leaking current alarm					*)
	MesFuse_Burned		: BOOL;		(* (NA) Power Distribution Unit Fuse Fail			*)
	MesOpen_CBBat		: BOOL;		(* (NA) Battery Switch Open							*)
	MesOpen_Aux			: BOOL;		(* (NA) LVDS Open Auxiliary contacts of contactor 	*)
	
	MesAlarmRectifer	: BOOL;		(* (NA) Rectifier failure							*)
	
END_STRUCT
END_TYPE

// ---- 01_Equipement_Library/UPS/UPS_PS10048.TcDUT
///////////
// Structure for PS100_48. Main operating data to be saved (ex:OPC).  
//////////
TYPE UPS_PS10048 :
STRUCT
		MesData             : UPS; 			(* MesData 																		*)
		                            		                                                                                
		MesSoc				: REAL; 		(* (%) Battery charge indicator 												*)
		MesUdc_48V			: REAL; 		(* (V) 48V output voltage 														*)
		MesUdc_12V			: REAL; 		(* (V) 12V output voltage 														*)
		MesUBatt			: REAL; 		(* (V) 12V battery voltage	    												*)
		MesIdc_12V			: REAL; 		(* (A) 12V output current 														*)
		MesIdc_Bat			: REAL;			(* (A) Battery current 															*)
		                            		                                                                                
		MesDischarge		: REAL; 		(* (V) Serious discharge threshold 												*)
		MesEbackUp			: REAL; 		(* (%) Energy backup threshold 	   												*)
		MesCapacity_Nom		: REAL; 		(* (Ah) NomCapa 				   												*)
		                                                                       												
		MesEBackUpEna		: BOOL;  		(* (Na) Energy backup enabled 	   												*)
		MesBatTestPer		: BOOL;  		(* (Na) Battery test period 	  												*)
		MesVacTripSelect	: BOOL;  		(* (NA) 0: Low. Off = 52Vac, Low = 129Vac. 1: High. Off = 69Vac, Low = 172Vac	*)
		                                                                                                                    
		MesToggleWrite		: BOOL;			(* (NA) Cal : True = read authorised  											*)
		MesToggleRead		: BOOL;			(* (NA) Cal : True = Write authorised 											*)
		                           		                                                                                    
		MesAlarm_AcOff		: BOOL;			(* (NA) True = AC off 															*)
		MesAlarm_GeneralOff	: BOOL;			(* (NA) True = Imminent shutdown 												*)
	//	MesAlarm_LowBat		: BOOL;			(* (NA) True = discharge 														*)
		MesAlarm_AcLow		: BOOL;			(* (NA) True = AC power supply low 												*)
		                                                                                                                    
		MesFault_Minor		: BOOL;			(* (NA) True = Minor fault (overtemp, overcurrent, overvolt) 					*)
		MesFault_Major		: BOOL;			(* (NA) True = Major fault : cannot recover 									*)
		MesFault_Bat		: BOOL;			(* (NA) True = Battery disconnected 											*)
		MesFault_Charger	: BOOL;			(* (NA) True = Charger out of order 											*)
		MesFault_12V		: BOOL;			(* (NA) True = 12V absent 														*)
		MesFault_48V		: BOOL;			(* (NA) True = 48V absent 														*)
		                           	
END_STRUCT
END_TYPE

// ---- 04_Application/COM/COM_Status.TcDUT
TYPE COM_Status :
	
// TO make it work, import the NetworkScan .exe, add it as a service and prepare the XML.

STRUCT
	// Network ( IP + port ) 
	MesWatchdog_Internet 		: BOOL := TRUE ; (* Watchdog internet    	   *)  
	MesWatchdog_Router 			: BOOL := TRUE ; (* Watchdog router      	   *) 
	MesWatchdog_Router_SMS  	: BOOL := TRUE ; (* Watchdog router SMS  	   *) 
	MesWatchdog_IndusPC 		: BOOL := TRUE ; (* Watchdog indusPC     	   *)  
	MesWatchdog_IEC104			: BOOL := TRUE ; (* Watchdog IEC104	     	   *) 
	MesWatchdog_PLC         	: BOOL := TRUE ; (* Watchdog PLC	     	   *) 

	
	// Services 
	MesRunning_HMIServer    	: BOOL :=TRUE  ; (* HMI server is running      *) 
	MesRunning_OpenVPN      	: BOOL :=TRUE  ; (* OpenVPN is running         *) 
	MesRunning_TV           	: BOOL :=TRUE  ; (* TV is running              *) 
	MesRunning_OPCUa        	: BOOL :=TRUE  ; (* OPC Ua is running          *) 
	MesRunning_Chronograf   	: BOOL :=TRUE  ; (* Chronograf is running      *) 
	MesRunning_Telegraf     	: BOOL :=TRUE  ; (* Telegraf is running        *) 
	MesRunning_Influx       	: BOOL :=TRUE  ; (* Influx is running          *) 
	MesRunning_ModBus       	: BOOL :=TRUE  ; (* Modbus TCP is running          *) 
	
END_STRUCT
END_TYPE

// ---- 04_Application/EMS/EMS.TcDUT
TYPE EMS :
STRUCT
	IN_EMS		: IN_EMS;
	OUT_EMS		: OUT_EMS;
	
	MesAlarmCode		: WORD;
	MesWarningCode		: WORD;
	
END_STRUCT
END_TYPE

// ---- 04_Application/EMS/IN_EMS.TcDUT
{attribute 'pack_mode' := '1'}
TYPE IN_EMS :
// Input for the SCADA
STRUCT
	
IN_Watchdog 						: REAL ; (* Value from EMS. Reinitializes to 1 at 1000. *)
IN_StateProduction 					: REAL ; (* Between the start of the montée and the end of the end of the pic du soir descente. "1" means True and "0" means False, pas utile pour le moment sur Janar mais je peux le garder au cas où*)
IN_SetptP_GRID_max 					: REAL ; (* Puissance max que l'on peut injecter sur le réseau*)
IN_SetptP_GRID_min 					: REAL ; (* Puissance min que l'on peut injecter sur le réseau*)
IN_SetptP_GRID						: REAL ; (* At Sub MV at Q100 power meter*)
IN_SetptShare_ESS1_PCS1 			: REAL ; (* Setpoint share between ESS1_PCS1, ESS1_PCS2, ESS2_PCS1, ESS2_PCS2, ESS3_PCS1 and ESS3_PCS2 at Sub MV*)
IN_CalCRateDischarge_ESS1_BAT1 		: REAL ; (* Average Discharge Crate of the year*)
IN_CalCRateCharge_ESS1_BAT1 		: REAL ; (* Average Charge Crate of the year*)
IN_CalRSoC_ESS1_BAT1 				: REAL ; (* Average rest SoC of the year*)
IN_CalCSoC_ESS1_BAT1 				: REAL ; (* Average center SoC of the year*)
IN_CalEnergyThroughput_ESS1_BAT1 	: REAL ; (* Energy throughput of the year*)
IN_CalPdc_ESS1_BAT1 				: REAL ; (* DC power of the year*)
IN_CalCRateDischarge_ESS1_BAT2		: REAL ; (* Average Discharge Crate of the year*)
IN_CalCRateCharge_ESS1_BAT2			: REAL ; (* Average Charge Crate of the year*)
IN_CalRSoC_ESS1_BAT2 				: REAL ; (* Average rest SoC of the year*)
IN_CalCSoC_ESS1_BAT2 				: REAL ; (* Average center SoC of the year*)
IN_CalEnergyThroughput_ESS1_BAT2 	: REAL ; (* Energy throughput of the year*)
IN_CalPdc_ESS1_BAT2 				: REAL ; (* DC power of the year*)

IN_TimeApplySetpoint_LINT           : LINT; (* EPOCH : Time at which the setpoint should be applied*)
END_STRUCT
END_TYPE

// ---- 04_Application/EMS/OUT_EMS.TcDUT
{attribute 'pack_mode' := '1'}
TYPE OUT_EMS :
// Output for the SCADA
STRUCT
	OUT_Watchdog 							: REAL ; (* Incremented value from EMS. Reinitializes to 1 at 1000. *)
	OUT_SetptP_GRID 						: REAL ; (* Setpoint received from Grid Manager*)
	OUT_MesP_GRID 							: REAL ; (* Average of previous minute (in Enercal-granularity sense) injected power*)
	OUT_CmdRebootEMS 						: BOOL ; (* Command the EMS to reboot : resets all parameters. "1" means True and "0" means False *)
	OUT_CmdKillEMS 							: BOOL ; (* Command the EMS to stop. "1" means True and "0" means False *)
	OUT_NoPenalties 						: BOOL ; (* There has been a Defaut GTE during production today. "1" means True and "0" means False. Pour le moment pas sûre que ça soit pertinent pour le CdC des AO CRE ZNI, à confirmer*)
	OUT_MesP_SPP 							: REAL ; (* At Sub MV (sum of the 2 SPPs), mean over the last minute*)
	OUT_MesAvailability_SPP 				: REAL ; (* Sum for the 2 SPPs : Pdc_Connected / Pdc_Tot for the inverters*)
	OUT_MesP_ESS 							: REAL ; (* At Sub MV (sum of the 2 PCSs)*)
	OUT_Balancing_SoC_Calibration_Required 	: BOOL;	(*(NA) Synthesis of the two Evnt01 signals for the EMS*)
	OUT_OngoingCalibration					: BOOL; (*(NA) SOC Calibration is ongoing (True) or NOT (False)*)
	OUT_Ecretage							: REAL;
END_STRUCT
END_TYPE

// ---- 04_Application/IO/IO.TcDUT
TYPE IO :
STRUCT
MesEventCode : ARRAY[1..7] OF WORD ; (*Akuo AlarmCode*)

END_STRUCT
END_TYPE

// ---- 04_Application/IO/ST_AI.TcDUT
{attribute 'OPC.UA.DA' := '1'}    
TYPE ST_AI :
STRUCT
		Value		  AT %I*	: INT	;
		Description 			: STRING	;

END_STRUCT
END_TYPE

// ---- 04_Application/IO/ST_AO.TcDUT
{attribute 'OPC.UA.DA' := '1'}    
TYPE ST_AO :
STRUCT
		Value		  AT %Q*	: INT	;
		Description 			: STRING	;

END_STRUCT
END_TYPE

// ---- 04_Application/IO/ST_DI.TcDUT
{attribute 'OPC.UA.DA' := '1'}    
TYPE ST_DI :
STRUCT
		Value		  AT %I*	: BOOL	;
		Description 			: STRING	;

END_STRUCT
END_TYPE

// ---- 04_Application/IO/ST_DO.TcDUT
{attribute 'OPC.UA.DA' := '1'}    
TYPE ST_DO :
STRUCT
		Value		  AT %Q*	: BOOL	;
		Description 			: STRING	;

END_STRUCT
END_TYPE

// ---- 04_Application/OPC/AllAlarms.TcDUT
TYPE AllAlarms :
STRUCT
PP_MesAlarmCode_1:BOOL ; 
PP_MesAlarmCode_2:BOOL ; 
PP_MesAlarmCode_3:BOOL ; 
PP_MesAlarmCode_4:BOOL ; 
PP_MesAlarmCode_5:BOOL ; 
PP_MesWarningCode_1:BOOL ; 
PP_MesWarningCode_2:BOOL ; 
PP_MesWarningCode_3:BOOL ; 
PP_MesWarningCode_5:BOOL ; 
PP_MesWarningCode_6:BOOL ; 
PP_MesWarningCode_7:BOOL ; 
PP_MesWarningCode_8:BOOL ; 
PP_MesWarningCode_9:BOOL ; 
PP_MesWarningCode_10:BOOL ; 
PP_MesWarningCode_12:BOOL ; 
PP_MesWarningCode_13:BOOL ; 
PP_MesWarningCode_14:BOOL ; 
PP_MesWarningCode_15:BOOL ; 
PP_MesWarningCode2_1:BOOL ; 
PP_MesWarningCode2_2:BOOL ; 
PP_MesWarningCode2_3:BOOL ; 
PP_MesWarningCode2_4:BOOL ; 
PP_MesWarningCode2_6:BOOL ; 
PP_MesWarningCode2_7:BOOL ; 
PP_MesWarningCode2_8:BOOL ; 
PP_MesWarningCode2_9:BOOL ; 
PP_MesWarningCode2_10:BOOL ; 
PP_MesWarningCode2_11:BOOL ; 
PP_MesWarningCode2_12:BOOL ; 
PP_MesWarningCode2_14:BOOL ; 
PP_MesEventCode_14:BOOL ; 
PP_MesEventCode_15:BOOL ; 



END_STRUCT
END_TYPE

// ---- 04_Application/OPC/AllDataR.TcDUT
TYPE AllDataR :
	
// 	REGLES : 														
// 	Mettre seulement les structures des produits 					
// 	Séparer les Structures (Pas AX_PTR mais PTR_1, PTR_2, ...)		
// 	Les noms des variables sont globales (Pas ION7650 mais PM) 		 
//	PP
//	PTR_1, PTR_2, PTR_3
//	INV		

STRUCT
	
//PP               	
	PP					: PP;              	   (* PP *)
	
//SUB_MV               	
	SUBMV				: SUBMV_Exd;       	   (* SUB.MV*)
//SUB_HV               	
	SUBHV				: SUBHV_Exd;       	   (* SUB.MV*)
// PTR        	
	PTR					: ARRAY[1..CstNbPTR_G] OF  PTR_Exd;        (* PTR *)



	ESS_Test			: ARRAY[1..CstNbPTR_G] OF  ESS_Exd;        (* PTR *)

	ESS					: ARRAY[1..CstNbPTR_G] OF  ESS_Exd;        (* PTR *)


	
//WS                	
	WS					: WS_RAV2;              		(* WS *)
                                           		
//COM                                      		
	SMS					: ServerSms;       		(* SMS      *)
	MAIL				: ServerMail;      		(* MAIL     *)
	COM					: COM_Status;	   		(* COM      *)
	CSV					: ServerCSV;       		(* CSV      *)
	CSVData				: LoggerCSV;       		(* CSVData  *) 
	OPCUA				: OPCAlarms ; 				(* OPCUA  *) 
	IO					: IO ; 	

END_STRUCT

END_TYPE

// ---- 04_Application/OPC/OPCAlarms.TcDUT
TYPE OPCAlarms :
	
// 	REGLES : 														
// 	Mettre seulement les structures des produits 					
// 	Séparer les Structures (Pas AX_PTR mais PTR_1, PTR_2, ...)		
// 	Les noms des variables sont globales (Pas ION7650 mais PM) 		 
//	PP
//	PTR_1, PTR_2, PTR_3
//	INV		

STRUCT
	
//OPC
	MesAlarmCode		: WORD ; 				 (* OPC Alarm Code   *)
	MesWarningCode		: WORD ; 				 (* OPC Warning Code *)
	MesEventCode 		: ARRAY[1..9] OF WORD ; (* OPC Event Code *)

END_STRUCT

END_TYPE

// ---- 04_Application/OPC/AllDataWPulse.TcDUT

TYPE AllDataWPulse :
STRUCT
	//Communication
	CmdReset_ServerSMS			: BOOL;			(* Reset SMS Server *)
	CmdReset_ServerMail			: BOOL;			(* Reset Mail server *)
	CmdReset_Router_ADSL		: BOOL;			(* Restart ADSL router *)	
	CmdReset_Router_4G			: BOOL;			(* Restart 4G router *)
	CmdReset_IPC				: BOOL;			(* Restart IPC *)
	CmdDeleteAllSms				: BOOL;  		(* Delete all SMS in the buffer *)
	CmdChangeInfos_PhoneEmail	: BOOL;			(* Apply new changes in Mail and SMS infos *)
	CmdReadInfosFromTarget_PhoneEmail	: BOOL ; 	(* Get Saved configuration *)
	CmdTestSms					: BOOL;         (* Test SMS function *)
	
	
	CmdRestart_OPCUA 	   		: BOOL;			(* Restart OPCUA *)
	CmdRestart_Teamviewer		: BOOL;			(* Restart Teamviewer *)
	CmdRestart_HMIServer 		: BOOL;			(* Restart HMIServer *)
	CmdRestart_Telegraf 			: BOOL;			(* Restart Codesys *)	


	CmdRestart_PLC				: BOOL;			(* Restart PLC *)
	CmdForcedStay_Connect		: BOOL;			(* Force the power plant to remains connected during a code restart or reboot *)
	CmdIpLauncher				: BOOL;			(* Get the public IP of the power plant	*)                  
	CmdStart_Vpn				: BOOL;			(* Start VPN *)
	CmdStop_Vpn					: BOOL;			(* Stop VPN *)
                         
	// Maintenance and Test     
	CmdInhibAllWrite			: BOOL; 		(* Force all digital and analog output to FALSE when activated. Inhibite communication write *) 
	CmdAllowAllWrite			: BOOL; 		(* Force all digital and analog output to TRUE when activated.  Allow communication write *)
	CmdInhibAllRead				: BOOL; 		(* Force all digital and analog input to FALSE when activated. Inhibite communication read *)
	CmdAllowAllRead				: BOOL; 		(* Force all digital and analog input to TRUE when activated. Allow communication read  *)
	CmdWriteSetptTanPhi			: BOOL; 		(* PP Setpoint TanphI *)
                           
	// SUB_MV                      
	CmdClose_MainMVCB			: BOOL; 		(* Close MainMVCB *)
	CmdOpen_MainMVCB			: BOOL;     	(* Open MainMVCB *)
	CmdReset_MainMVCB			: BOOL;     	(* Reset MainMVCB *)	

	CmdOpen_FeederMVCB			: ARRAY[1..CstNbFeederMVCB_G] OF  BOOL;     (* Open FeederMVCB [ARRAY]*)
	CmdClose_FeederMVCB			: ARRAY[1..CstNbFeederMVCB_G] OF  BOOL;   	(* Close FeederMVCB [ARRAY]*)
	CmdReset_FeederMVCB			: ARRAY[1..CstNbFeederMVCB_G] OF  BOOL;   	(* Reset FeederMVCB [ARRAY]*)
	                                        
	CmdStartLocalSetptP_PP		: BOOL;     	(*	Activate local setpoint at substation *)
	CmdStopLocalSetptP_PP		: BOOL;     	(*	Desactivate local setpoint at substation *)
	
	// PTR
		CmdOpen_PTR					: ARRAY[1..CstNbPTR_G] OF BOOL;		(*	Open corresponding PTR [ARRAY]*) 
		CmdClose_PTR				: ARRAY[1..CstNbPTR_G] OF BOOL;		(* Close corresponding PTR [ARRAY]*)
	
	// Inverter
		CmdStart_INV				: ARRAY[1..CstNbPTR_G] OF ARRAY[1..CstNbInv_PTR_G] OF BOOL;		(* Switch On inverter [ARRAY]*)
		CmdStop_INV					: ARRAY[1..CstNbPTR_G] OF ARRAY[1..CstNbInv_PTR_G] OF BOOL;     (* Switch Off inverter [ARRAY]*)
		CmdStartSetptP_INV			: ARRAY[1..CstNbPTR_G] OF ARRAY[1..CstNbInv_PTR_G] OF BOOL;     (* Activate local setpoint on inverter [ARRAY]*)
		CmdStopSetptP_INV			: ARRAY[1..CstNbPTR_G] OF ARRAY[1..CstNbInv_PTR_G] OF BOOL;		(* Desactivate local setpoint on inverter [ARRAY]*)
		CmdToggleCom_Read			: ARRAY[1..CstNbPTR_G] OF ARRAY[1..CstNbInv_PTR_G] OF BOOL;		(* Inverter Toggle Read Communication [ARRAY]*) 
		CmdToggleCom_Write			: ARRAY[1..CstNbPTR_G] OF ARRAY[1..CstNbInv_PTR_G] OF BOOL;		(* Inverter Toggle Write Communication [ARRAY]*)
	
	// PCS
		CmdReset_ESS					: ARRAY[1..CstNbESS_G] OF BOOL;		(* Reset ESS [ARRAY]*)
		CmdCalibrationCalculation_PCS	: ARRAY[1..CstNbESS_G] OF ARRAY[1..CstNbPcs_ESS_G] OF BOOL;		(* Calibrate calculation PCS [ARRAY]*)
		CmdStart_PCS					: ARRAY[1..CstNbESS_G] OF ARRAY[1..CstNbPcs_ESS_G] OF BOOL;		(* Switch On PCS [ARRAY]*)
		CmdStop_PCS						: ARRAY[1..CstNbESS_G] OF ARRAY[1..CstNbPcs_ESS_G] OF BOOL;     (* Switch Off PCS [ARRAY]*)
		CmdStandby_PCS					: ARRAY[1..CstNbESS_G] OF ARRAY[1..CstNbPcs_ESS_G] OF BOOL;     (* Switch to standby PCS [ARRAY]*)
		CmdReset_PCS					: ARRAY[1..CstNbESS_G] OF ARRAY[1..CstNbPcs_ESS_G] OF BOOL;     (* Reset PCS [ARRAY]*)
		CmdLocal_PCS					: ARRAY[1..CstNbESS_G] OF ARRAY[1..CstNbPcs_ESS_G] OF BOOL;		(* Switch PCS to local [ARRAY]*)
		
	// BAT
		CmdOpenDc_BAT					: ARRAY[1..CstNbESS_G] OF ARRAY[1..CstNbBat_ESS_G] OF BOOL;		(* Open DC Battery [ARRAY]*) 
		CmdCloseDc_BAT					: ARRAY[1..CstNbESS_G] OF ARRAY[1..CstNbBat_ESS_G] OF BOOL;		(* Close DC Battery [ARRAY]*) 
		CmdReset_BAT					: ARRAY[1..CstNbESS_G] OF ARRAY[1..CstNbBat_ESS_G] OF BOOL;		(* Reset Battery [ARRAY]*) 
		
	// UPS 
		CmdRestart_UPS48			: BOOL ; (*	Restart UPS *)
		CmdRestart_UPS24			: BOOL ; (*	Restart UPS *)
	
	// SD
		CmdReset_SD					: BOOL; (* Reset all Smoke detectors with one commande*)
	
